LIN {X 0,Y 432.342,Z 838.796,A -85,B 0,C 180,E1 21138.258,E2 21138.258} C_VEL
LIN {X 0,Y 432.858,Z 830.958,A -85,B 0,C 180,E1 21135.431,E2 21135.431} C_VEL
LIN {X 0,Y 433.67,Z 821.606,A -85,B 0,C 180,E1 21132.698,E2 21132.698} C_VEL
LIN {X 0,Y 434.794,Z 810.85,A -85,B 0,C 180,E1 21130.103,E2 21130.103} C_VEL
LIN {X 0,Y 436.206,Z 798.707,A -85,B 0,C 180,E1 21127.636,E2 21127.636} C_VEL
LIN {X 0,Y 437.923,Z 785.326,A -85,B 0,C 180,E1 21125.304,E2 21125.304} C_VEL
LIN {X 0,Y 439.952,Z 770.003,A -85,B 0,C 180,E1 21123.039,E2 21123.039} C_VEL
LIN {X 0,Y 442.141,Z 753.688,A -85,B 0,C 180,E1 21120.984,E2 21120.984} C_VEL
LIN {X 0,Y 444.605,Z 735.27,A -85,B 0,C 180,E1 21119.004,E2 21119.004} C_VEL
LIN {X 0,Y 447.006,Z 716.668,A -85,B 0,C 180,E1 21117.305,E2 21117.305} C_VEL
LIN {X 0,Y 449.34,Z 697.148,A -85,B 0,C 180,E1 21115.817,E2 21115.817} C_VEL
LIN {X 0,Y 451.636,Z 676.412,A -85,B 0,C 180,E1 21114.499,E2 21114.499} C_VEL
LIN {X 0,Y 453.72,Z 655.392,A -85,B 0,C 180,E1 21113.41,E2 21113.41} C_VEL
LIN {X 0,Y 455.533,Z 633.906,A -85,B 0,C 180,E1 21112.542,E2 21112.542} C_VEL
LIN {X 0,Y 456.937,Z 612.319,A -85,B 0,C 180,E1 21111.907,E2 21111.907} C_VEL
LIN {X 0,Y 458.017,Z 582.765,A -85,B 0,C 180,E1 21111.317,E2 21111.317} C_VEL
LIN {X 0,Y 464.099,Z 362.571,A -85,B 0,C 180,E1 21107.412,E2 21107.412} C_VEL
LIN {X 0,Y 464.742,Z 333.232,A -85,B 0,C 180,E1 21106.874,E2 21106.874} C_VEL
LIN {X 0,Y 464.066,Z 331.268,A -85,B 0,C 180,E1 21106.761,E2 21106.761} C_VEL
LIN {X 0,Y 451.341,Z 310.172,A -85,B 0,C 180,E1 21104.898,E2 21104.898} C_VEL
LIN {X 0,Y 448.432,Z 305.591,A -85,B 0,C 180,E1 21104.436,E2 21104.436} C_VEL
LIN {X 0,Y 441.155,Z 290.184,A -85,B 0,C 180,E1 21101.959,E2 21101.959} C_VEL
LIN {X 0,Y 437.067,Z 281.96,A -85,B 0,C 180,E1 21100.518,E2 21100.518} C_VEL
LIN {X 0,Y 434.855,Z 277.707,A -85,B 0,C 180,E1 21099.732,E2 21099.732} C_VEL
LIN {X 0,Y 433.312,Z 274.093,A -85,B 0,C 180,E1 21099.045,E2 21099.045} C_VEL
LIN {X 0,Y 433.24,Z 273.726,A -85,B 0,C 180,E1 21097.204,E2 21097.204} C_VEL
LIN {X 0,Y 433.217,Z 273.762,A -85,B 0,C 180,E1 21093.477,E2 21093.477} C_VEL
LIN {X 0,Y 433.2,Z 273.744,A -85,B 0,C 180,E1 21089.751,E2 21089.751} C_VEL
LIN {X 0,Y 433.199,Z 273.765,A -85,B 0,C 180,E1 21086.01,E2 21086.01} C_VEL
LIN {X 0,Y 433.212,Z 273.763,A -85,B 0,C 180,E1 21082.384,E2 21082.384} C_VEL
LIN {X 0,Y 433.236,Z 273.758,A -85,B 0,C 180,E1 21078.711,E2 21078.711} C_VEL
LIN {X 0,Y 433.233,Z 273.756,A -85,B 0,C 180,E1 21074.843,E2 21074.843} C_VEL
LIN {X 0,Y 433.21,Z 273.757,A -85,B 0,C 180,E1 21071.044,E2 21071.044} C_VEL
LIN {X 0,Y 433.19,Z 273.76,A -85,B 0,C 180,E1 21067.426,E2 21067.426} C_VEL
LIN {X 0,Y 433.193,Z 273.766,A -85,B 0,C 180,E1 21063.705,E2 21063.705} C_VEL
LIN {X 0,Y 433.208,Z 273.769,A -85,B 0,C 180,E1 21060,E2 21060} C_VEL
LIN {X 0,Y 433.236,Z 273.77,A -85,B 0,C 180,E1 21056.295,E2 21056.295} C_VEL
LIN {X 0,Y 433.261,Z 273.765,A -85,B 0,C 180,E1 21052.441,E2 21052.441} C_VEL
LIN {X 0,Y 433.254,Z 273.759,A -85,B 0,C 180,E1 21048.552,E2 21048.552} C_VEL
LIN {X 0,Y 433.255,Z 273.755,A -85,B 0,C 180,E1 21044.715,E2 21044.715} C_VEL
LIN {X 0,Y 433.234,Z 273.756,A -85,B 0,C 180,E1 21041.009,E2 21041.009} C_VEL
LIN {X 0,Y 433.226,Z 273.756,A -85,B 0,C 180,E1 21037.33,E2 21037.33} C_VEL
LIN {X 0,Y 433.232,Z 273.757,A -85,B 0,C 180,E1 21033.549,E2 21033.549} C_VEL
LIN {X 0,Y 433.252,Z 273.729,A -85,B 0,C 180,E1 21029.928,E2 21029.928} C_VEL
LIN {X 0,Y 433.259,Z 273.766,A -85,B 0,C 180,E1 21026.049,E2 21026.049} C_VEL
LIN {X 0,Y 433.251,Z 273.723,A -85,B 0,C 180,E1 21022.297,E2 21022.297} C_VEL
LIN {X 0,Y 433.255,Z 273.731,A -85,B 0,C 180,E1 21018.522,E2 21018.522} C_VEL
LIN {X 0,Y 433.329,Z 274.222,A -85,B 0,C 180,E1 21017.773,E2 21017.773} C_VEL
LIN {X 0,Y 434.815,Z 277.61,A -85,B 0,C 180,E1 21017.105,E2 21017.105} C_VEL
LIN {X 0,Y 441.185,Z 290.862,A -85,B 0,C 180,E1 21014.631,E2 21014.631} C_VEL
LIN {X 0,Y 448.978,Z 308.721,A -85,B 0,C 180,E1 21011.656,E2 21011.656} C_VEL
LIN {X 0,Y 455.647,Z 325.683,A -85,B 0,C 180,E1 21009.149,E2 21009.149} C_VEL
LIN {X 0,Y 461.307,Z 360.167,A -85,B 0,C 180,E1 21007.848,E2 21007.848} C_VEL
LIN {X 0,Y 457.058,Z 564.663,A -85,B 0,C 180,E1 21004.513,E2 21004.513} C_VEL
LIN {X 0,Y 456.111,Z 572.366,A -85,B 0,C 180,E1 21004.467,E2 21004.467} C_VEL
LIN {X 0,Y 450.547,Z 592.852,A -85,B 0,C 180,E1 21004.59,E2 21004.59} C_VEL
LIN {X 0,Y 449.686,Z 599.4,A -85,B 0,C 180,E1 21004.491,E2 21004.491} C_VEL
LIN {X 0,Y 448.443,Z 619.453,A -85,B 0,C 180,E1 21003.895,E2 21003.895} C_VEL
LIN {X 0,Y 446.74,Z 639.526,A -85,B 0,C 180,E1 21003.061,E2 21003.061} C_VEL
LIN {X 0,Y 444.586,Z 659.236,A -85,B 0,C 180,E1 21001.98,E2 21001.98} C_VEL
LIN {X 0,Y 442.233,Z 677.397,A -85,B 0,C 180,E1 21000.728,E2 21000.728} C_VEL
LIN {X 0,Y 439.717,Z 694.787,A -85,B 0,C 180,E1 20999.266,E2 20999.266} C_VEL
LIN {X 0,Y 437.101,Z 711.358,A -85,B 0,C 180,E1 20997.594,E2 20997.594} C_VEL
LIN {X 0,Y 434.515,Z 726.984,A -85,B 0,C 180,E1 20995.709,E2 20995.709} C_VEL
LIN {X 0,Y 431.994,Z 741.73,A -85,B 0,C 180,E1 20993.573,E2 20993.573} C_VEL
LIN {X 0,Y 429.869,Z 754.225,A -85,B 0,C 180,E1 20991.418,E2 20991.418} C_VEL
LIN {X 0,Y 427.951,Z 766.244,A -85,B 0,C 180,E1 20988.95,E2 20988.95} C_VEL
LIN {X 0,Y 426.43,Z 776.74,A -85,B 0,C 180,E1 20986.341,E2 20986.341} C_VEL
LIN {X 0,Y 425.369,Z 785.323,A -85,B 0,C 180,E1 20983.733,E2 20983.733} C_VEL
LIN {X 0,Y 424.64,Z 792.647,A -85,B 0,C 180,E1 20980.926,E2 20980.926} C_VEL
LIN {X 0,Y 424.24,Z 798.109,A -85,B 0,C 180,E1 20978.129,E2 20978.129} C_VEL
LIN {X 0,Y 424.047,Z 801.843,A -85,B 0,C 180,E1 20975.412,E2 20975.412} C_VEL
LIN {X 0,Y 423.984,Z 804.16,A -85,B 0,C 180,E1 20972.568,E2 20972.568} C_VEL
LIN {X 0,Y 423.977,Z 804.889,A -85,B 0,C 180,E1 20969.865,E2 20969.865} C_VEL
LIN {X 0,Y 423.986,Z 804.012,A -85,B 0,C 180,E1 20967.026,E2 20967.026} C_VEL
LIN {X 0,Y 424.055,Z 801.599,A -85,B 0,C 180,E1 20964.278,E2 20964.278} C_VEL
LIN {X 0,Y 424.272,Z 797.547,A -85,B 0,C 180,E1 20961.462,E2 20961.462} C_VEL
LIN {X 0,Y 424.687,Z 792.034,A -85,B 0,C 180,E1 20958.732,E2 20958.732} C_VEL
LIN {X 0,Y 425.429,Z 784.801,A -85,B 0,C 180,E1 20955.991,E2 20955.991} C_VEL
LIN {X 0,Y 426.596,Z 775.591,A -85,B 0,C 180,E1 20953.245,E2 20953.245} C_VEL
LIN {X 0,Y 428.083,Z 765.421,A -85,B 0,C 180,E1 20950.773,E2 20950.773} C_VEL
LIN {X 0,Y 429.914,Z 753.959,A -85,B 0,C 180,E1 20948.441,E2 20948.441} C_VEL
LIN {X 0,Y 432.079,Z 741.214,A -85,B 0,C 180,E1 20946.257,E2 20946.257} C_VEL
LIN {X 0,Y 434.58,Z 726.625,A -85,B 0,C 180,E1 20944.152,E2 20944.152} C_VEL
LIN {X 0,Y 437.285,Z 710.326,A -85,B 0,C 180,E1 20942.197,E2 20942.197} C_VEL
LIN {X 0,Y 439.941,Z 693.383,A -85,B 0,C 180,E1 20940.511,E2 20940.511} C_VEL
LIN {X 0,Y 442.454,Z 675.834,A -85,B 0,C 180,E1 20939.063,E2 20939.063} C_VEL
LIN {X 0,Y 444.822,Z 657.259,A -85,B 0,C 180,E1 20937.811,E2 20937.811} C_VEL
LIN {X 0,Y 446.807,Z 638.92,A -85,B 0,C 180,E1 20936.818,E2 20936.818} C_VEL
LIN {X 0,Y 448.538,Z 618.51,A -85,B 0,C 180,E1 20935.979,E2 20935.979} C_VEL
LIN {X 0,Y 449.739,Z 598.65,A -85,B 0,C 180,E1 20935.398,E2 20935.398} C_VEL
LIN {X 0,Y 450.572,Z 571.156,A -85,B 0,C 180,E1 20934.885,E2 20934.885} C_VEL
LIN {X 0,Y 455.175,Z 360.498,A -85,B 0,C 180,E1 20931.4,E2 20931.4} C_VEL
LIN {X 0,Y 449.82,Z 329.343,A -85,B 0,C 180,E1 20930.173,E2 20930.173} C_VEL
LIN {X 0,Y 447.126,Z 324.378,A -85,B 0,C 180,E1 20929.689,E2 20929.689} C_VEL
LIN {X 0,Y 440.044,Z 306.845,A -85,B 0,C 180,E1 20926.929,E2 20926.929} C_VEL
LIN {X 0,Y 433.12,Z 291.369,A -85,B 0,C 180,E1 20924.201,E2 20924.201} C_VEL
LIN {X 0,Y 428.555,Z 282.138,A -85,B 0,C 180,E1 20922.397,E2 20922.397} C_VEL
LIN {X 0,Y 426.709,Z 278.339,A -85,B 0,C 180,E1 20921.63,E2 20921.63} C_VEL
LIN {X 0,Y 425.329,Z 274.888,A -85,B 0,C 180,E1 20920.864,E2 20920.864} C_VEL
LIN {X 0,Y 425.309,Z 274.709,A -85,B 0,C 180,E1 20917.162,E2 20917.162} C_VEL
LIN {X 0,Y 425.316,Z 274.741,A -85,B 0,C 180,E1 20913.374,E2 20913.374} C_VEL
LIN {X 0,Y 425.317,Z 274.725,A -85,B 0,C 180,E1 20909.566,E2 20909.566} C_VEL
LIN {X 0,Y 425.318,Z 274.743,A -85,B 0,C 180,E1 20905.78,E2 20905.78} C_VEL
LIN {X 0,Y 425.314,Z 274.743,A -85,B 0,C 180,E1 20901.95,E2 20901.95} C_VEL
LIN {X 0,Y 425.292,Z 274.744,A -85,B 0,C 180,E1 20898.221,E2 20898.221} C_VEL
LIN {X 0,Y 425.282,Z 274.743,A -85,B 0,C 180,E1 20894.395,E2 20894.395} C_VEL
LIN {X 0,Y 425.278,Z 274.742,A -85,B 0,C 180,E1 20890.567,E2 20890.567} C_VEL
LIN {X 0,Y 425.28,Z 274.748,A -85,B 0,C 180,E1 20886.751,E2 20886.751} C_VEL
LIN {X 0,Y 425.289,Z 274.754,A -85,B 0,C 180,E1 20882.965,E2 20882.965} C_VEL
LIN {X 0,Y 425.307,Z 274.759,A -85,B 0,C 180,E1 20879.192,E2 20879.192} C_VEL
LIN {X 0,Y 425.304,Z 274.757,A -85,B 0,C 180,E1 20875.28,E2 20875.28} C_VEL
LIN {X 0,Y 425.293,Z 274.751,A -85,B 0,C 180,E1 20871.483,E2 20871.483} C_VEL
LIN {X 0,Y 425.27,Z 274.749,A -85,B 0,C 180,E1 20867.646,E2 20867.646} C_VEL
LIN {X 0,Y 425.241,Z 274.748,A -85,B 0,C 180,E1 20864.032,E2 20864.032} C_VEL
LIN {X 0,Y 425.247,Z 274.75,A -85,B 0,C 180,E1 20860.21,E2 20860.21} C_VEL
LIN {X 0,Y 425.256,Z 274.752,A -85,B 0,C 180,E1 20856.441,E2 20856.441} C_VEL
LIN {X 0,Y 425.28,Z 274.753,A -85,B 0,C 180,E1 20852.707,E2 20852.707} C_VEL
LIN {X 0,Y 425.309,Z 274.707,A -85,B 0,C 180,E1 20849.013,E2 20849.013} C_VEL
LIN {X 0,Y 425.312,Z 274.742,A -85,B 0,C 180,E1 20845.128,E2 20845.128} C_VEL
LIN {X 0,Y 425.305,Z 274.978,A -85,B 0,C 180,E1 20842.151,E2 20842.151} C_VEL
LIN {X 0,Y 426.746,Z 278.433,A -85,B 0,C 180,E1 20841.448,E2 20841.448} C_VEL
LIN {X 0,Y 427.86,Z 280.355,A -85,B 0,C 180,E1 20841.052,E2 20841.052} C_VEL
LIN {X 0,Y 434.06,Z 292.497,A -85,B 0,C 180,E1 20838.792,E2 20838.792} C_VEL
LIN {X 0,Y 440.782,Z 306.575,A -85,B 0,C 180,E1 20836.47,E2 20836.47} C_VEL
LIN {X 0,Y 453.474,Z 326.821,A -85,B 0,C 180,E1 20834.498,E2 20834.498} C_VEL
LIN {X 0,Y 458.777,Z 336.288,A -85,B 0,C 180,E1 20833.704,E2 20833.704} C_VEL
LIN {X 0,Y 452.487,Z 549.122,A -85,B 0,C 180,E1 20829.882,E2 20829.882} C_VEL
LIN {X 0,Y 450.683,Z 607.462,A -85,B 0,C 180,E1 20828.803,E2 20828.803} C_VEL
LIN {X 0,Y 449.222,Z 629.594,A -85,B 0,C 180,E1 20828.179,E2 20828.179} C_VEL
LIN {X 0,Y 447.415,Z 650.894,A -85,B 0,C 180,E1 20827.351,E2 20827.351} C_VEL
LIN {X 0,Y 445.277,Z 671.891,A -85,B 0,C 180,E1 20826.307,E2 20826.307} C_VEL
LIN {X 0,Y 442.975,Z 691.862,A -85,B 0,C 180,E1 20825.067,E2 20825.067} C_VEL
LIN {X 0,Y 440.506,Z 711.034,A -85,B 0,C 180,E1 20823.629,E2 20823.629} C_VEL
LIN {X 0,Y 437.891,Z 730.422,A -85,B 0,C 180,E1 20821.91,E2 20821.91} C_VEL
LIN {X 0,Y 435.415,Z 748.423,A -85,B 0,C 180,E1 20820.036,E2 20820.036} C_VEL
LIN {X 0,Y 432.988,Z 765.307,A -85,B 0,C 180,E1 20817.954,E2 20817.954} C_VEL
LIN {X 0,Y 430.798,Z 780.808,A -85,B 0,C 180,E1 20815.722,E2 20815.722} C_VEL
LIN {X 0,Y 429.003,Z 794.229,A -85,B 0,C 180,E1 20813.486,E2 20813.486} C_VEL
LIN {X 0,Y 427.37,Z 806.957,A -85,B 0,C 180,E1 20810.974,E2 20810.974} C_VEL
LIN {X 0,Y 426.071,Z 818.284,A -85,B 0,C 180,E1 20808.328,E2 20808.328} C_VEL
LIN {X 0,Y 425.154,Z 827.798,A -85,B 0,C 180,E1 20805.691,E2 20805.691} C_VEL
LIN {X 0,Y 424.519,Z 835.821,A -85,B 0,C 180,E1 20802.929,E2 20802.929} C_VEL
LIN {X 0,Y 424.146,Z 842.478,A -85,B 0,C 180,E1 20800.046,E2 20800.046} C_VEL
LIN {X 0,Y 423.986,Z 847.207,A -85,B 0,C 180,E1 20797.316,E2 20797.316} C_VEL
LIN {X 0,Y 423.922,Z 850.344,A -85,B 0,C 180,E1 20794.599,E2 20794.599} C_VEL
LIN {X 0,Y 423.903,Z 852.117,A -85,B 0,C 180,E1 20791.892,E2 20791.892} C_VEL
LIN {X 0,Y 423.905,Z 852.344,A -85,B 0,C 180,E1 20789.189,E2 20789.189} C_VEL
LIN {X 0,Y 423.911,Z 851.265,A -85,B 0,C 180,E1 20786.484,E2 20786.484} C_VEL
LIN {X 0,Y 423.945,Z 848.609,A -85,B 0,C 180,E1 20783.772,E2 20783.772} C_VEL
LIN {X 0,Y 424.056,Z 844.592,A -85,B 0,C 180,E1 20781.048,E2 20781.048} C_VEL
LIN {X 0,Y 424.332,Z 838.905,A -85,B 0,C 180,E1 20778.309,E2 20778.309} C_VEL
LIN {X 0,Y 424.859,Z 831.189,A -85,B 0,C 180,E1 20775.416,E2 20775.416} C_VEL
LIN {X 0,Y 425.69,Z 822.043,A -85,B 0,C 180,E1 20772.645,E2 20772.645} C_VEL
LIN {X 0,Y 426.888,Z 811.022,A -85,B 0,C 180,E1 20769.921,E2 20769.921} C_VEL
LIN {X 0,Y 428.404,Z 798.659,A -85,B 0,C 180,E1 20767.351,E2 20767.351} C_VEL
LIN {X 0,Y 430.206,Z 785.265,A -85,B 0,C 180,E1 20764.977,E2 20764.977} C_VEL
LIN {X 0,Y 432.265,Z 770.439,A -85,B 0,C 180,E1 20762.744,E2 20762.744} C_VEL
LIN {X 0,Y 434.634,Z 753.687,A -85,B 0,C 180,E1 20760.585,E2 20760.585} C_VEL
LIN {X 0,Y 437.135,Z 736.043,A -85,B 0,C 180,E1 20758.645,E2 20758.645} C_VEL
LIN {X 0,Y 439.757,Z 716.905,A -85,B 0,C 180,E1 20756.852,E2 20756.852} C_VEL
LIN {X 0,Y 442.22,Z 697.805,A -85,B 0,C 180,E1 20755.353,E2 20755.353} C_VEL
LIN {X 0,Y 444.704,Z 676.971,A -85,B 0,C 180,E1 20753.99,E2 20753.99} C_VEL
LIN {X 0,Y 446.923,Z 656.118,A -85,B 0,C 180,E1 20752.881,E2 20752.881} C_VEL
LIN {X 0,Y 448.807,Z 634.988,A -85,B 0,C 180,E1 20752.008,E2 20752.008} C_VEL
LIN {X 0,Y 450.335,Z 613.288,A -85,B 0,C 180,E1 20751.347,E2 20751.347} C_VEL
LIN {X 0,Y 451.401,Z 587.981,A -85,B 0,C 180,E1 20750.816,E2 20750.816} C_VEL
LIN {X 0,Y 457.893,Z 365.769,A -85,B 0,C 180,E1 20746.824,E2 20746.824} C_VEL
LIN {X 0,Y 458.663,Z 335.761,A -85,B 0,C 180,E1 20746.273,E2 20746.273} C_VEL
LIN {X 0,Y 446.377,Z 315.309,A -85,B 0,C 180,E1 20744.425,E2 20744.425} C_VEL
LIN {X 0,Y 440.405,Z 305.946,A -85,B 0,C 180,E1 20743.464,E2 20743.464} C_VEL
LIN {X 0,Y 433.548,Z 291.624,A -85,B 0,C 180,E1 20741.052,E2 20741.052} C_VEL
LIN {X 0,Y 428.845,Z 282.534,A -85,B 0,C 180,E1 20739.358,E2 20739.358} C_VEL
LIN {X 0,Y 427.13,Z 278.929,A -85,B 0,C 180,E1 20738.683,E2 20738.683} C_VEL
LIN {X 0,Y 425.432,Z 275.615,A -85,B 0,C 180,E1 20738.007,E2 20738.007} C_VEL
LIN {X 0,Y 425.301,Z 274.942,A -85,B 0,C 180,E1 20737.824,E2 20737.824} C_VEL
LIN {X 0,Y 425.283,Z 274.761,A -85,B 0,C 180,E1 20734.35,E2 20734.35} C_VEL
LIN {X 0,Y 425.296,Z 274.711,A -85,B 0,C 180,E1 20730.635,E2 20730.635} C_VEL
LIN {X 0,Y 425.308,Z 274.746,A -85,B 0,C 180,E1 20726.832,E2 20726.832} C_VEL
LIN {X 0,Y 425.299,Z 274.745,A -85,B 0,C 180,E1 20722.97,E2 20722.97} C_VEL
LIN {X 0,Y 425.268,Z 274.746,A -85,B 0,C 180,E1 20719.217,E2 20719.217} C_VEL
LIN {X 0,Y 425.244,Z 274.747,A -85,B 0,C 180,E1 20715.548,E2 20715.548} C_VEL
LIN {X 0,Y 425.241,Z 274.748,A -85,B 0,C 180,E1 20711.804,E2 20711.804} C_VEL
LIN {X 0,Y 425.26,Z 274.752,A -85,B 0,C 180,E1 20708.11,E2 20708.11} C_VEL
LIN {X 0,Y 425.294,Z 274.755,A -85,B 0,C 180,E1 20704.449,E2 20704.449} C_VEL
LIN {X 0,Y 425.313,Z 274.757,A -85,B 0,C 180,E1 20700.539,E2 20700.539} C_VEL
LIN {X 0,Y 425.308,Z 274.757,A -85,B 0,C 180,E1 20696.63,E2 20696.63} C_VEL
LIN {X 0,Y 425.314,Z 274.75,A -85,B 0,C 180,E1 20692.707,E2 20692.707} C_VEL
LIN {X 0,Y 425.296,Z 274.745,A -85,B 0,C 180,E1 20688.885,E2 20688.885} C_VEL
LIN {X 0,Y 425.282,Z 274.744,A -85,B 0,C 180,E1 20685.151,E2 20685.151} C_VEL
LIN {X 0,Y 425.284,Z 274.744,A -85,B 0,C 180,E1 20681.341,E2 20681.341} C_VEL
LIN {X 0,Y 425.287,Z 274.744,A -85,B 0,C 180,E1 20677.467,E2 20677.467} C_VEL
LIN {X 0,Y 425.296,Z 274.744,A -85,B 0,C 180,E1 20673.619,E2 20673.619} C_VEL
LIN {X 0,Y 425.311,Z 274.714,A -85,B 0,C 180,E1 20669.894,E2 20669.894} C_VEL
LIN {X 0,Y 425.317,Z 274.756,A -85,B 0,C 180,E1 20665.978,E2 20665.978} C_VEL
LIN {X 0,Y 425.313,Z 274.711,A -85,B 0,C 180,E1 20662.151,E2 20662.151} C_VEL
LIN {X 0,Y 425.338,Z 274.956,A -85,B 0,C 180,E1 20658.987,E2 20658.987} C_VEL
LIN {X 0,Y 426.671,Z 278.285,A -85,B 0,C 180,E1 20658.277,E2 20658.277} C_VEL
LIN {X 0,Y 431.664,Z 288.3,A -85,B 0,C 180,E1 20656.275,E2 20656.275} C_VEL
LIN {X 0,Y 438.677,Z 303.743,A -85,B 0,C 180,E1 20653.497,E2 20653.497} C_VEL
LIN {X 0,Y 445.468,Z 320.179,A -85,B 0,C 180,E1 20650.852,E2 20650.852} C_VEL
LIN {X 0,Y 447.868,Z 326.008,A -85,B 0,C 180,E1 20650.027,E2 20650.027} C_VEL
LIN {X 0,Y 450.129,Z 330.276,A -85,B 0,C 180,E1 20649.675,E2 20649.675} C_VEL
LIN {X 0,Y 455.193,Z 361.696,A -85,B 0,C 180,E1 20648.477,E2 20648.477} C_VEL
LIN {X 0,Y 449.956,Z 594.214,A -85,B 0,C 180,E1 20644.617,E2 20644.617} C_VEL
LIN {X 0,Y 449.686,Z 599.4,A -85,B 0,C 180,E1 20644.491,E2 20644.491} C_VEL
LIN {X 0,Y 448.171,Z 608.086,A -85,B 0,C 180,E1 20644.363,E2 20644.363} C_VEL
LIN {X 0,Y 442.571,Z 625.029,A -85,B 0,C 180,E1 20644.211,E2 20644.211} C_VEL
LIN {X 0,Y 440.918,Z 632.44,A -85,B 0,C 180,E1 20643.996,E2 20643.996} C_VEL
LIN {X 0,Y 440.796,Z 633.461,A -85,B 0,C 180,E1 20643.953,E2 20643.953} C_VEL
LIN {X 0,Y 438.804,Z 652.395,A -85,B 0,C 180,E1 20642.995,E2 20642.995} C_VEL
LIN {X 0,Y 436.421,Z 671.242,A -85,B 0,C 180,E1 20641.79,E2 20641.79} C_VEL
LIN {X 0,Y 433.688,Z 689.657,A -85,B 0,C 180,E1 20640.324,E2 20640.324} C_VEL
LIN {X 0,Y 430.962,Z 706.412,A -85,B 0,C 180,E1 20638.701,E2 20638.701} C_VEL
LIN {X 0,Y 428.095,Z 722.858,A -85,B 0,C 180,E1 20636.792,E2 20636.792} C_VEL
LIN {X 0,Y 425.43,Z 737.71,A -85,B 0,C 180,E1 20634.729,E2 20634.729} C_VEL
LIN {X 0,Y 423.03,Z 751.127,A -85,B 0,C 180,E1 20632.513,E2 20632.513} C_VEL
LIN {X 0,Y 420.834,Z 763.774,A -85,B 0,C 180,E1 20630.006,E2 20630.006} C_VEL
LIN {X 0,Y 419.054,Z 774.772,A -85,B 0,C 180,E1 20627.352,E2 20627.352} C_VEL
LIN {X 0,Y 417.782,Z 783.758,A -85,B 0,C 180,E1 20624.695,E2 20624.695} C_VEL
LIN {X 0,Y 416.886,Z 791.376,A -85,B 0,C 180,E1 20621.888,E2 20621.888} C_VEL
LIN {X 0,Y 416.366,Z 797.415,A -85,B 0,C 180,E1 20618.98,E2 20618.98} C_VEL
LIN {X 0,Y 416.119,Z 801.567,A -85,B 0,C 180,E1 20616.207,E2 20616.207} C_VEL
LIN {X 0,Y 416.009,Z 804.256,A -85,B 0,C 180,E1 20613.307,E2 20613.307} C_VEL
LIN {X 0,Y 415.982,Z 805.258,A -85,B 0,C 180,E1 20610.551,E2 20610.551} C_VEL
LIN {X 0,Y 415.992,Z 804.785,A -85,B 0,C 180,E1 20607.658,E2 20607.658} C_VEL
LIN {X 0,Y 416.059,Z 802.871,A -85,B 0,C 180,E1 20604.899,E2 20604.899} C_VEL
LIN {X 0,Y 416.248,Z 799.229,A -85,B 0,C 180,E1 20601.992,E2 20601.992} C_VEL
LIN {X 0,Y 416.638,Z 794.079,A -85,B 0,C 180,E1 20599.212,E2 20599.212} C_VEL
LIN {X 0,Y 417.349,Z 787.26,A -85,B 0,C 180,E1 20596.422,E2 20596.422} C_VEL
LIN {X 0,Y 418.488,Z 778.588,A -85,B 0,C 180,E1 20593.625,E2 20593.625} C_VEL
LIN {X 0,Y 420.053,Z 768.416,A -85,B 0,C 180,E1 20590.968,E2 20590.968} C_VEL
LIN {X 0,Y 422.031,Z 756.769,A -85,B 0,C 180,E1 20588.456,E2 20588.456} C_VEL
LIN {X 0,Y 424.425,Z 743.434,A -85,B 0,C 180,E1 20586.072,E2 20586.072} C_VEL
LIN {X 0,Y 427.061,Z 728.752,A -85,B 0,C 180,E1 20583.887,E2 20583.887} C_VEL
LIN {X 0,Y 429.773,Z 713.364,A -85,B 0,C 180,E1 20581.97,E2 20581.97} C_VEL
LIN {X 0,Y 432.621,Z 696.412,A -85,B 0,C 180,E1 20580.206,E2 20580.206} C_VEL
LIN {X 0,Y 435.317,Z 678.927,A -85,B 0,C 180,E1 20578.697,E2 20578.697} C_VEL
LIN {X 0,Y 437.856,Z 660.443,A -85,B 0,C 180,E1 20577.391,E2 20577.391} C_VEL
LIN {X 0,Y 440.031,Z 641.486,A -85,B 0,C 180,E1 20576.33,E2 20576.33} C_VEL
LIN {X 0,Y 441.83,Z 621.78,A -85,B 0,C 180,E1 20575.477,E2 20575.477} C_VEL
LIN {X 0,Y 443.254,Z 600.889,A -85,B 0,C 180,E1 20574.828,E2 20574.828} C_VEL
LIN {X 0,Y 444.096,Z 578.129,A -85,B 0,C 180,E1 20574.37,E2 20574.37} C_VEL
LIN {X 0,Y 449.135,Z 362.019,A -85,B 0,C 180,E1 20570.754,E2 20570.754} C_VEL
LIN {X 0,Y 444.346,Z 333.544,A -85,B 0,C 180,E1 20569.613,E2 20569.613} C_VEL
LIN {X 0,Y 439.058,Z 324.277,A -85,B 0,C 180,E1 20568.721,E2 20568.721} C_VEL
LIN {X 0,Y 432.276,Z 307.715,A -85,B 0,C 180,E1 20566.001,E2 20566.001} C_VEL
LIN {X 0,Y 425.286,Z 292.398,A -85,B 0,C 180,E1 20563.169,E2 20563.169} C_VEL
LIN {X 0,Y 420.839,Z 283.447,A -85,B 0,C 180,E1 20561.338,E2 20561.338} C_VEL
LIN {X 0,Y 418.859,Z 279.471,A -85,B 0,C 180,E1 20560.489,E2 20560.489} C_VEL
LIN {X 0,Y 417.4,Z 275.929,A -85,B 0,C 180,E1 20559.677,E2 20559.677} C_VEL
LIN {X 0,Y 417.375,Z 275.708,A -85,B 0,C 180,E1 20555.935,E2 20555.935} C_VEL
LIN {X 0,Y 417.371,Z 275.697,A -85,B 0,C 180,E1 20552.129,E2 20552.129} C_VEL
LIN {X 0,Y 417.367,Z 275.747,A -85,B 0,C 180,E1 20548.316,E2 20548.316} C_VEL
LIN {X 0,Y 417.357,Z 275.748,A -85,B 0,C 180,E1 20544.448,E2 20544.448} C_VEL
LIN {X 0,Y 417.354,Z 275.749,A -85,B 0,C 180,E1 20540.62,E2 20540.62} C_VEL
LIN {X 0,Y 417.349,Z 275.75,A -85,B 0,C 180,E1 20536.708,E2 20536.708} C_VEL
LIN {X 0,Y 417.353,Z 275.747,A -85,B 0,C 180,E1 20532.874,E2 20532.874} C_VEL
LIN {X 0,Y 417.363,Z 275.736,A -85,B 0,C 180,E1 20529.098,E2 20529.098} C_VEL
LIN {X 0,Y 417.374,Z 275.729,A -85,B 0,C 180,E1 20525.361,E2 20525.361} C_VEL
LIN {X 0,Y 417.369,Z 275.729,A -85,B 0,C 180,E1 20521.51,E2 20521.51} C_VEL
LIN {X 0,Y 417.34,Z 275.737,A -85,B 0,C 180,E1 20517.803,E2 20517.803} C_VEL
LIN {X 0,Y 417.321,Z 275.749,A -85,B 0,C 180,E1 20514.087,E2 20514.087} C_VEL
LIN {X 0,Y 417.311,Z 275.752,A -85,B 0,C 180,E1 20510.345,E2 20510.345} C_VEL
LIN {X 0,Y 417.311,Z 275.752,A -85,B 0,C 180,E1 20506.561,E2 20506.561} C_VEL
LIN {X 0,Y 417.329,Z 275.749,A -85,B 0,C 180,E1 20502.861,E2 20502.861} C_VEL
LIN {X 0,Y 417.359,Z 275.745,A -85,B 0,C 180,E1 20499.087,E2 20499.087} C_VEL
LIN {X 0,Y 417.363,Z 275.749,A -85,B 0,C 180,E1 20495.214,E2 20495.214} C_VEL
LIN {X 0,Y 417.371,Z 275.741,A -85,B 0,C 180,E1 20491.255,E2 20491.255} C_VEL
LIN {X 0,Y 417.346,Z 275.708,A -85,B 0,C 180,E1 20487.488,E2 20487.488} C_VEL
LIN {X 0,Y 417.338,Z 275.74,A -85,B 0,C 180,E1 20483.718,E2 20483.718} C_VEL
LIN {X 0,Y 417.47,Z 276.341,A -85,B 0,C 180,E1 20483.266,E2 20483.266} C_VEL
LIN {X 0,Y 419.119,Z 279.84,A -85,B 0,C 180,E1 20482.531,E2 20482.531} C_VEL
LIN {X 0,Y 422.59,Z 286.572,A -85,B 0,C 180,E1 20481.171,E2 20481.171} C_VEL
LIN {X 0,Y 428.388,Z 297.927,A -85,B 0,C 180,E1 20479.016,E2 20479.016} C_VEL
LIN {X 0,Y 432.651,Z 306.855,A -85,B 0,C 180,E1 20477.511,E2 20477.511} C_VEL
LIN {X 0,Y 445.037,Z 326.238,A -85,B 0,C 180,E1 20475.496,E2 20475.496} C_VEL
LIN {X 0,Y 452.67,Z 339.479,A -85,B 0,C 180,E1 20474.315,E2 20474.315} C_VEL
LIN {X 0,Y 446.088,Z 550.51,A -85,B 0,C 180,E1 20470.48,E2 20470.48} C_VEL
LIN {X 0,Y 444.229,Z 607.33,A -85,B 0,C 180,E1 20469.413,E2 20469.413} C_VEL
LIN {X 0,Y 442.691,Z 629.472,A -85,B 0,C 180,E1 20468.782,E2 20468.782} C_VEL
LIN {X 0,Y 440.763,Z 651.005,A -85,B 0,C 180,E1 20467.933,E2 20467.933} C_VEL
LIN {X 0,Y 438.557,Z 671.563,A -85,B 0,C 180,E1 20466.896,E2 20466.896} C_VEL
LIN {X 0,Y 436.072,Z 691.87,A -85,B 0,C 180,E1 20465.618,E2 20465.618} C_VEL
LIN {X 0,Y 433.479,Z 710.831,A -85,B 0,C 180,E1 20464.169,E2 20464.169} C_VEL
LIN {X 0,Y 430.704,Z 730.058,A -85,B 0,C 180,E1 20462.428,E2 20462.428} C_VEL
LIN {X 0,Y 427.965,Z 748.573,A -85,B 0,C 180,E1 20460.447,E2 20460.447} C_VEL
LIN {X 0,Y 425.274,Z 766.36,A -85,B 0,C 180,E1 20458.2,E2 20458.2} C_VEL
LIN {X 0,Y 422.994,Z 781.631,A -85,B 0,C 180,E1 20455.931,E2 20455.931} C_VEL
LIN {X 0,Y 421.016,Z 795.593,A -85,B 0,C 180,E1 20453.514,E2 20453.514} C_VEL
LIN {X 0,Y 419.36,Z 808.181,A -85,B 0,C 180,E1 20450.955,E2 20450.955} C_VEL
LIN {X 0,Y 418.042,Z 819.255,A -85,B 0,C 180,E1 20448.259,E2 20448.259} C_VEL
LIN {X 0,Y 417.081,Z 828.917,A -85,B 0,C 180,E1 20445.432,E2 20445.432} C_VEL
LIN {X 0,Y 416.464,Z 836.753,A -85,B 0,C 180,E1 20442.619,E2 20442.619} C_VEL
LIN {X 0,Y 416.13,Z 842.766,A -85,B 0,C 180,E1 20439.822,E2 20439.822} C_VEL
LIN {X 0,Y 415.977,Z 847.473,A -85,B 0,C 180,E1 20436.902,E2 20436.902} C_VEL
LIN {X 0,Y 415.926,Z 850.236,A -85,B 0,C 180,E1 20434.274,E2 20434.274} C_VEL
LIN {X 0,Y 415.916,Z 851.802,A -85,B 0,C 180,E1 20431.377,E2 20431.377} C_VEL
LIN {X 0,Y 415.919,Z 851.826,A -85,B 0,C 180,E1 20428.76,E2 20428.76} C_VEL
LIN {X 0,Y 415.923,Z 850.354,A -85,B 0,C 180,E1 20425.864,E2 20425.864} C_VEL
LIN {X 0,Y 415.968,Z 847.638,A -85,B 0,C 180,E1 20423.236,E2 20423.236} C_VEL
LIN {X 0,Y 416.121,Z 843.039,A -85,B 0,C 180,E1 20420.317,E2 20420.317} C_VEL
LIN {X 0,Y 416.443,Z 837.104,A -85,B 0,C 180,E1 20417.521,E2 20417.521} C_VEL
LIN {X 0,Y 417.042,Z 829.343,A -85,B 0,C 180,E1 20414.709,E2 20414.709} C_VEL
LIN {X 0,Y 417.986,Z 819.796,A -85,B 0,C 180,E1 20411.883,E2 20411.883} C_VEL
LIN {X 0,Y 419.28,Z 808.837,A -85,B 0,C 180,E1 20409.187,E2 20409.187} C_VEL
LIN {X 0,Y 420.911,Z 796.348,A -85,B 0,C 180,E1 20406.629,E2 20406.629} C_VEL
LIN {X 0,Y 422.995,Z 781.648,A -85,B 0,C 180,E1 20404.069,E2 20404.069} C_VEL
LIN {X 0,Y 425.276,Z 766.368,A -85,B 0,C 180,E1 20401.8,E2 20401.8} C_VEL
LIN {X 0,Y 427.966,Z 748.572,A -85,B 0,C 180,E1 20399.552,E2 20399.552} C_VEL
LIN {X 0,Y 430.705,Z 730.059,A -85,B 0,C 180,E1 20397.572,E2 20397.572} C_VEL
LIN {X 0,Y 433.479,Z 710.833,A -85,B 0,C 180,E1 20395.831,E2 20395.831} C_VEL
LIN {X 0,Y 436.191,Z 690.835,A -85,B 0,C 180,E1 20394.313,E2 20394.313} C_VEL
LIN {X 0,Y 438.756,Z 670.028,A -85,B 0,C 180,E1 20393.015,E2 20393.015} C_VEL
LIN {X 0,Y 440.986,Z 648.747,A -85,B 0,C 180,E1 20391.966,E2 20391.966} C_VEL
LIN {X 0,Y 442.902,Z 626.421,A -85,B 0,C 180,E1 20391.12,E2 20391.12} C_VEL
LIN {X 0,Y 444.377,Z 604.158,A -85,B 0,C 180,E1 20390.521,E2 20390.521} C_VEL
LIN {X 0,Y 450.904,Z 395.819,A -85,B 0,C 180,E1 20386.708,E2 20386.708} C_VEL
LIN {X 0,Y 452.564,Z 339.015,A -85,B 0,C 180,E1 20385.665,E2 20385.665} C_VEL
LIN {X 0,Y 440.669,Z 319.242,A -85,B 0,C 180,E1 20383.819,E2 20383.819} C_VEL
LIN {X 0,Y 432.233,Z 306.09,A -85,B 0,C 180,E1 20382.4,E2 20382.4} C_VEL
LIN {X 0,Y 425.42,Z 292.132,A -85,B 0,C 180,E1 20379.913,E2 20379.913} C_VEL
LIN {X 0,Y 421.536,Z 284.405,A -85,B 0,C 180,E1 20378.422,E2 20378.422} C_VEL
LIN {X 0,Y 418.695,Z 279.242,A -85,B 0,C 180,E1 20377.341,E2 20377.341} C_VEL
LIN {X 0,Y 417.39,Z 275.942,A -85,B 0,C 180,E1 20376.618,E2 20376.618} C_VEL
LIN {X 0,Y 417.371,Z 275.714,A -85,B 0,C 180,E1 20372.943,E2 20372.943} C_VEL
LIN {X 0,Y 417.36,Z 275.731,A -85,B 0,C 180,E1 20369.099,E2 20369.099} C_VEL
LIN {X 0,Y 417.332,Z 275.747,A -85,B 0,C 180,E1 20365.395,E2 20365.395} C_VEL
LIN {X 0,Y 417.315,Z 275.751,A -85,B 0,C 180,E1 20361.628,E2 20361.628} C_VEL
LIN {X 0,Y 417.308,Z 275.751,A -85,B 0,C 180,E1 20357.859,E2 20357.859} C_VEL
LIN {X 0,Y 417.308,Z 275.752,A -85,B 0,C 180,E1 20353.989,E2 20353.989} C_VEL
LIN {X 0,Y 417.324,Z 275.746,A -85,B 0,C 180,E1 20350.212,E2 20350.212} C_VEL
LIN {X 0,Y 417.353,Z 275.735,A -85,B 0,C 180,E1 20346.465,E2 20346.465} C_VEL
LIN {X 0,Y 417.362,Z 275.731,A -85,B 0,C 180,E1 20342.609,E2 20342.609} C_VEL
LIN {X 0,Y 417.364,Z 275.73,A -85,B 0,C 180,E1 20338.764,E2 20338.764} C_VEL
LIN {X 0,Y 417.353,Z 275.735,A -85,B 0,C 180,E1 20334.914,E2 20334.914} C_VEL
LIN {X 0,Y 417.341,Z 275.746,A -85,B 0,C 180,E1 20331.18,E2 20331.18} C_VEL
LIN {X 0,Y 417.336,Z 275.75,A -85,B 0,C 180,E1 20327.407,E2 20327.407} C_VEL
LIN {X 0,Y 417.344,Z 275.748,A -85,B 0,C 180,E1 20323.578,E2 20323.578} C_VEL
LIN {X 0,Y 417.351,Z 275.747,A -85,B 0,C 180,E1 20319.673,E2 20319.673} C_VEL
LIN {X 0,Y 417.367,Z 275.746,A -85,B 0,C 180,E1 20315.883,E2 20315.883} C_VEL
LIN {X 0,Y 417.381,Z 275.745,A -85,B 0,C 180,E1 20311.996,E2 20311.996} C_VEL
LIN {X 0,Y 417.375,Z 275.691,A -85,B 0,C 180,E1 20308.195,E2 20308.195} C_VEL
LIN {X 0,Y 417.376,Z 275.715,A -85,B 0,C 180,E1 20304.3,E2 20304.3} C_VEL
LIN {X 0,Y 417.388,Z 275.793,A -85,B 0,C 180,E1 20300.416,E2 20300.416} C_VEL
LIN {X 0,Y 417.49,Z 276.399,A -85,B 0,C 180,E1 20300.07,E2 20300.07} C_VEL
LIN {X 0,Y 419.009,Z 279.686,A -85,B 0,C 180,E1 20299.349,E2 20299.349} C_VEL
LIN {X 0,Y 424.057,Z 289.852,A -85,B 0,C 180,E1 20297.23,E2 20297.23} C_VEL
LIN {X 0,Y 431.015,Z 304.881,A -85,B 0,C 180,E1 20294.398,E2 20294.398} C_VEL
LIN {X 0,Y 438.144,Z 322,A -85,B 0,C 180,E1 20291.538,E2 20291.538} C_VEL
LIN {X 0,Y 439.835,Z 325.908,A -85,B 0,C 180,E1 20290.999,E2 20290.999} C_VEL
LIN {X 0,Y 444.608,Z 334.386,A -85,B 0,C 180,E1 20290.24,E2 20290.24} C_VEL
LIN {X 0,Y 449.133,Z 363.266,A -85,B 0,C 180,E1 20289.122,E2 20289.122} C_VEL
LIN {X 0,Y 443.581,Z 594.524,A -85,B 0,C 180,E1 20285.237,E2 20285.237} C_VEL
LIN {X 0,Y 442.379,Z 614.806,A -85,B 0,C 180,E1 20284.675,E2 20284.675} C_VEL
LIN {X 0,Y 440.796,Z 633.461,A -85,B 0,C 180,E1 20283.953,E2 20283.953} C_VEL
LIN {X 0,Y 439.234,Z 640.947,A -85,B 0,C 180,E1 20283.687,E2 20283.687} C_VEL
LIN {X 0,Y 432.206,Z 659.277,A -85,B 0,C 180,E1 20283.137,E2 20283.137} C_VEL
LIN {X 0,Y 430.464,Z 666.153,A -85,B 0,C 180,E1 20282.76,E2 20282.76} C_VEL
LIN {X 0,Y 427.832,Z 684.074,A -85,B 0,C 180,E1 20281.409,E2 20281.409} C_VEL
LIN {X 0,Y 424.994,Z 701.253,A -85,B 0,C 180,E1 20279.839,E2 20279.839} C_VEL
LIN {X 0,Y 421.977,Z 718.025,A -85,B 0,C 180,E1 20277.979,E2 20277.979} C_VEL
LIN {X 0,Y 419.09,Z 733.175,A -85,B 0,C 180,E1 20275.962,E2 20275.962} C_VEL
LIN {X 0,Y 416.466,Z 746.908,A -85,B 0,C 180,E1 20273.786,E2 20273.786} C_VEL
LIN {X 0,Y 414.067,Z 759.647,A -85,B 0,C 180,E1 20271.384,E2 20271.384} C_VEL
LIN {X 0,Y 412.066,Z 770.942,A -85,B 0,C 180,E1 20268.827,E2 20268.827} C_VEL
LIN {X 0,Y 410.484,Z 780.762,A -85,B 0,C 180,E1 20266.121,E2 20266.121} C_VEL
LIN {X 0,Y 409.332,Z 789.057,A -85,B 0,C 180,E1 20263.274,E2 20263.274} C_VEL
LIN {X 0,Y 408.623,Z 795.53,A -85,B 0,C 180,E1 20260.432,E2 20260.432} C_VEL
LIN {X 0,Y 408.226,Z 800.544,A -85,B 0,C 180,E1 20257.458,E2 20257.458} C_VEL
LIN {X 0,Y 408.062,Z 803.752,A -85,B 0,C 180,E1 20254.638,E2 20254.638} C_VEL
LIN {X 0,Y 408.006,Z 805.449,A -85,B 0,C 180,E1 20251.826,E2 20251.826} C_VEL
LIN {X 0,Y 407.999,Z 805.657,A -85,B 0,C 180,E1 20249.017,E2 20249.017} C_VEL
LIN {X 0,Y 408.036,Z 804.357,A -85,B 0,C 180,E1 20246.066,E2 20246.066} C_VEL
LIN {X 0,Y 408.168,Z 801.645,A -85,B 0,C 180,E1 20243.248,E2 20243.248} C_VEL
LIN {X 0,Y 408.493,Z 797.096,A -85,B 0,C 180,E1 20240.277,E2 20240.277} C_VEL
LIN {X 0,Y 409.094,Z 791.054,A -85,B 0,C 180,E1 20237.437,E2 20237.437} C_VEL
LIN {X 0,Y 410.104,Z 783.251,A -85,B 0,C 180,E1 20234.589,E2 20234.589} C_VEL
LIN {X 0,Y 411.623,Z 773.473,A -85,B 0,C 180,E1 20231.739,E2 20231.739} C_VEL
LIN {X 0,Y 413.501,Z 762.75,A -85,B 0,C 180,E1 20229.18,E2 20229.18} C_VEL
LIN {X 0,Y 415.848,Z 750.273,A -85,B 0,C 180,E1 20226.705,E2 20226.705} C_VEL
LIN {X 0,Y 418.552,Z 736.183,A -85,B 0,C 180,E1 20224.382,E2 20224.382} C_VEL
LIN {X 0,Y 421.329,Z 721.469,A -85,B 0,C 180,E1 20222.359,E2 20222.359} C_VEL
LIN {X 0,Y 424.267,Z 705.296,A -85,B 0,C 180,E1 20220.493,E2 20220.493} C_VEL
LIN {X 0,Y 427.299,Z 687.408,A -85,B 0,C 180,E1 20218.783,E2 20218.783} C_VEL
LIN {X 0,Y 429.932,Z 670.252,A -85,B 0,C 180,E1 20217.428,E2 20217.428} C_VEL
LIN {X 0,Y 432.443,Z 651.32,A -85,B 0,C 180,E1 20216.217,E2 20216.217} C_VEL
LIN {X 0,Y 434.475,Z 632.614,A -85,B 0,C 180,E1 20215.281,E2 20215.281} C_VEL
LIN {X 0,Y 436.223,Z 612.023,A -85,B 0,C 180,E1 20214.502,E2 20214.502} C_VEL
LIN {X 0,Y 437.392,Z 591.49,A -85,B 0,C 180,E1 20213.966,E2 20213.966} C_VEL
LIN {X 0,Y 443.15,Z 363.519,A -85,B 0,C 180,E1 20210.091,E2 20210.091} C_VEL
LIN {X 0,Y 438.84,Z 337.569,A -85,B 0,C 180,E1 20209.026,E2 20209.026} C_VEL
LIN {X 0,Y 431.082,Z 324.339,A -85,B 0,C 180,E1 20207.723,E2 20207.723} C_VEL
LIN {X 0,Y 424.021,Z 307.59,A -85,B 0,C 180,E1 20204.834,E2 20204.834} C_VEL
LIN {X 0,Y 417.38,Z 293.285,A -85,B 0,C 180,E1 20202.046,E2 20202.046} C_VEL
LIN {X 0,Y 413.208,Z 284.897,A -85,B 0,C 180,E1 20200.246,E2 20200.246} C_VEL
LIN {X 0,Y 410.943,Z 280.475,A -85,B 0,C 180,E1 20199.243,E2 20199.243} C_VEL
LIN {X 0,Y 409.463,Z 276.928,A -85,B 0,C 180,E1 20198.388,E2 20198.388} C_VEL
LIN {X 0,Y 409.428,Z 276.732,A -85,B 0,C 180,E1 20194.681,E2 20194.681} C_VEL
LIN {X 0,Y 409.418,Z 276.68,A -85,B 0,C 180,E1 20190.691,E2 20190.691} C_VEL
LIN {X 0,Y 409.423,Z 276.725,A -85,B 0,C 180,E1 20186.859,E2 20186.859} C_VEL
LIN {X 0,Y 409.424,Z 276.722,A -85,B 0,C 180,E1 20182.979,E2 20182.979} C_VEL
LIN {X 0,Y 409.426,Z 276.721,A -85,B 0,C 180,E1 20179.08,E2 20179.08} C_VEL
LIN {X 0,Y 409.431,Z 276.72,A -85,B 0,C 180,E1 20175.148,E2 20175.148} C_VEL
LIN {X 0,Y 409.434,Z 276.722,A -85,B 0,C 180,E1 20171.266,E2 20171.266} C_VEL
LIN {X 0,Y 409.44,Z 276.727,A -85,B 0,C 180,E1 20167.296,E2 20167.296} C_VEL
LIN {X 0,Y 409.432,Z 276.735,A -85,B 0,C 180,E1 20163.36,E2 20163.36} C_VEL
LIN {X 0,Y 409.439,Z 276.734,A -85,B 0,C 180,E1 20159.441,E2 20159.441} C_VEL
LIN {X 0,Y 409.418,Z 276.732,A -85,B 0,C 180,E1 20155.518,E2 20155.518} C_VEL
LIN {X 0,Y 409.397,Z 276.729,A -85,B 0,C 180,E1 20151.715,E2 20151.715} C_VEL
LIN {X 0,Y 409.378,Z 276.725,A -85,B 0,C 180,E1 20147.875,E2 20147.875} C_VEL
LIN {X 0,Y 409.362,Z 276.724,A -85,B 0,C 180,E1 20144.124,E2 20144.124} C_VEL
LIN {X 0,Y 409.37,Z 276.725,A -85,B 0,C 180,E1 20140.303,E2 20140.303} C_VEL
LIN {X 0,Y 409.384,Z 276.727,A -85,B 0,C 180,E1 20136.541,E2 20136.541} C_VEL
LIN {X 0,Y 409.405,Z 276.729,A -85,B 0,C 180,E1 20132.741,E2 20132.741} C_VEL
LIN {X 0,Y 409.427,Z 276.68,A -85,B 0,C 180,E1 20128.984,E2 20128.984} C_VEL
LIN {X 0,Y 409.439,Z 276.763,A -85,B 0,C 180,E1 20124.979,E2 20124.979} C_VEL
LIN {X 0,Y 409.499,Z 277.282,A -85,B 0,C 180,E1 20124.58,E2 20124.58} C_VEL
LIN {X 0,Y 410.902,Z 280.472,A -85,B 0,C 180,E1 20123.886,E2 20123.886} C_VEL
LIN {X 0,Y 412.233,Z 282.702,A -85,B 0,C 180,E1 20123.369,E2 20123.369} C_VEL
LIN {X 0,Y 417.123,Z 292.223,A -85,B 0,C 180,E1 20121.39,E2 20121.39} C_VEL
LIN {X 0,Y 422.919,Z 303.865,A -85,B 0,C 180,E1 20119.158,E2 20119.158} C_VEL
LIN {X 0,Y 424.91,Z 307.634,A -85,B 0,C 180,E1 20118.54,E2 20118.54} C_VEL
LIN {X 0,Y 437.673,Z 327.267,A -85,B 0,C 180,E1 20116.377,E2 20116.377} C_VEL
LIN {X 0,Y 446.618,Z 342.628,A -85,B 0,C 180,E1 20114.943,E2 20114.943} C_VEL
LIN {X 0,Y 439.729,Z 552.46,A -85,B 0,C 180,E1 20111.085,E2 20111.085} C_VEL
LIN {X 0,Y 437.831,Z 607.289,A -85,B 0,C 180,E1 20110.041,E2 20110.041} C_VEL
LIN {X 0,Y 436.214,Z 629.437,A -85,B 0,C 180,E1 20109.402,E2 20109.402} C_VEL
LIN {X 0,Y 434.228,Z 650.557,A -85,B 0,C 180,E1 20108.561,E2 20108.561} C_VEL
LIN {X 0,Y 431.902,Z 671.271,A -85,B 0,C 180,E1 20107.505,E2 20107.505} C_VEL
LIN {X 0,Y 429.233,Z 691.872,A -85,B 0,C 180,E1 20106.192,E2 20106.192} C_VEL
LIN {X 0,Y 426.384,Z 711.572,A -85,B 0,C 180,E1 20104.655,E2 20104.655} C_VEL
LIN {X 0,Y 423.354,Z 731.258,A -85,B 0,C 180,E1 20102.82,E2 20102.82} C_VEL
LIN {X 0,Y 420.495,Z 749.333,A -85,B 0,C 180,E1 20100.824,E2 20100.824} C_VEL
LIN {X 0,Y 417.73,Z 766.44,A -85,B 0,C 180,E1 20098.6,E2 20098.6} C_VEL
LIN {X 0,Y 415.333,Z 781.572,A -85,B 0,C 180,E1 20096.292,E2 20096.292} C_VEL
LIN {X 0,Y 413.141,Z 796.223,A -85,B 0,C 180,E1 20093.686,E2 20093.686} C_VEL
LIN {X 0,Y 411.414,Z 808.789,A -85,B 0,C 180,E1 20091.056,E2 20091.056} C_VEL
LIN {X 0,Y 410.068,Z 819.639,A -85,B 0,C 180,E1 20088.332,E2 20088.332} C_VEL
LIN {X 0,Y 409.082,Z 829.168,A -85,B 0,C 180,E1 20085.45,E2 20085.45} C_VEL
LIN {X 0,Y 408.457,Z 836.891,A -85,B 0,C 180,E1 20082.583,E2 20082.583} C_VEL
LIN {X 0,Y 408.125,Z 842.797,A -85,B 0,C 180,E1 20079.732,E2 20079.732} C_VEL
LIN {X 0,Y 407.975,Z 847.332,A -85,B 0,C 180,E1 20076.756,E2 20076.756} C_VEL
LIN {X 0,Y 407.932,Z 850.015,A -85,B 0,C 180,E1 20074.076,E2 20074.076} C_VEL
LIN {X 0,Y 407.933,Z 851.401,A -85,B 0,C 180,E1 20071.124,E2 20071.124} C_VEL
LIN {X 0,Y 407.925,Z 851.328,A -85,B 0,C 180,E1 20068.455,E2 20068.455} C_VEL
LIN {X 0,Y 407.939,Z 849.658,A -85,B 0,C 180,E1 20065.502,E2 20065.502} C_VEL
LIN {X 0,Y 407.995,Z 846.656,A -85,B 0,C 180,E1 20062.679,E2 20062.679} C_VEL
LIN {X 0,Y 408.159,Z 842,A -85,B 0,C 180,E1 20059.841,E2 20059.841} C_VEL
LIN {X 0,Y 408.557,Z 835.469,A -85,B 0,C 180,E1 20056.845,E2 20056.845} C_VEL
LIN {X 0,Y 409.242,Z 827.465,A -85,B 0,C 180,E1 20053.974,E2 20053.974} C_VEL
LIN {X 0,Y 410.248,Z 818.029,A -85,B 0,C 180,E1 20051.234,E2 20051.234} C_VEL
LIN {X 0,Y 411.7,Z 806.612,A -85,B 0,C 180,E1 20048.459,E2 20048.459} C_VEL
LIN {X 0,Y 413.482,Z 794.012,A -85,B 0,C 180,E1 20045.88,E2 20045.88} C_VEL
LIN {X 0,Y 415.612,Z 779.791,A -85,B 0,C 180,E1 20043.419,E2 20043.419} C_VEL
LIN {X 0,Y 418.218,Z 763.265,A -85,B 0,C 180,E1 20040.967,E2 20040.967} C_VEL
LIN {X 0,Y 420.977,Z 746.317,A -85,B 0,C 180,E1 20038.818,E2 20038.818} C_VEL
LIN {X 0,Y 423.86,Z 728.205,A -85,B 0,C 180,E1 20036.868,E2 20036.868} C_VEL
LIN {X 0,Y 426.749,Z 709.062,A -85,B 0,C 180,E1 20035.133,E2 20035.133} C_VEL
LIN {X 0,Y 429.717,Z 688.098,A -85,B 0,C 180,E1 20033.553,E2 20033.553} C_VEL
LIN {X 0,Y 432.358,Z 667.587,A -85,B 0,C 180,E1 20032.29,E2 20032.29} C_VEL
LIN {X 0,Y 434.547,Z 647.452,A -85,B 0,C 180,E1 20031.299,E2 20031.299} C_VEL
LIN {X 0,Y 436.501,Z 625.542,A -85,B 0,C 180,E1 20030.472,E2 20030.472} C_VEL
LIN {X 0,Y 438.045,Z 602.78,A -85,B 0,C 180,E1 20029.865,E2 20029.865} C_VEL
LIN {X 0,Y 444.965,Z 392.608,A -85,B 0,C 180,E1 20025.975,E2 20025.975} C_VEL
LIN {X 0,Y 446.516,Z 342.285,A -85,B 0,C 180,E1 20025.04,E2 20025.04} C_VEL
LIN {X 0,Y 434.279,Z 321.944,A -85,B 0,C 180,E1 20023.073,E2 20023.073} C_VEL
LIN {X 0,Y 424.163,Z 306.39,A -85,B 0,C 180,E1 20021.302,E2 20021.302} C_VEL
LIN {X 0,Y 418.035,Z 293.983,A -85,B 0,C 180,E1 20018.979,E2 20018.979} C_VEL
LIN {X 0,Y 413.537,Z 285.26,A -85,B 0,C 180,E1 20017.189,E2 20017.189} C_VEL
LIN {X 0,Y 411.569,Z 281.281,A -85,B 0,C 180,E1 20016.353,E2 20016.353} C_VEL
LIN {X 0,Y 409.782,Z 278.351,A -85,B 0,C 180,E1 20015.66,E2 20015.66} C_VEL
LIN {X 0,Y 409.444,Z 276.933,A -85,B 0,C 180,E1 20015.313,E2 20015.313} C_VEL
LIN {X 0,Y 409.392,Z 276.684,A -85,B 0,C 180,E1 20011.51,E2 20011.51} C_VEL
LIN {X 0,Y 409.385,Z 276.74,A -85,B 0,C 180,E1 20007.806,E2 20007.806} C_VEL
LIN {X 0,Y 409.378,Z 276.732,A -85,B 0,C 180,E1 20003.918,E2 20003.918} C_VEL
LIN {X 0,Y 409.381,Z 276.727,A -85,B 0,C 180,E1 20000.143,E2 20000.143} C_VEL
LIN {X 0,Y 409.385,Z 276.725,A -85,B 0,C 180,E1 19996.312,E2 19996.312} C_VEL
LIN {X 0,Y 409.405,Z 276.727,A -85,B 0,C 180,E1 19992.554,E2 19992.554} C_VEL
LIN {X 0,Y 409.417,Z 276.73,A -85,B 0,C 180,E1 19988.567,E2 19988.567} C_VEL
LIN {X 0,Y 409.422,Z 276.734,A -85,B 0,C 180,E1 19984.622,E2 19984.622} C_VEL
LIN {X 0,Y 409.433,Z 276.738,A -85,B 0,C 180,E1 19980.699,E2 19980.699} C_VEL
LIN {X 0,Y 409.422,Z 276.733,A -85,B 0,C 180,E1 19976.78,E2 19976.78} C_VEL
LIN {X 0,Y 409.423,Z 276.726,A -85,B 0,C 180,E1 19972.845,E2 19972.845} C_VEL
LIN {X 0,Y 409.409,Z 276.721,A -85,B 0,C 180,E1 19969.018,E2 19969.018} C_VEL
LIN {X 0,Y 409.401,Z 276.72,A -85,B 0,C 180,E1 19965.263,E2 19965.263} C_VEL
LIN {X 0,Y 409.406,Z 276.721,A -85,B 0,C 180,E1 19961.341,E2 19961.341} C_VEL
LIN {X 0,Y 409.41,Z 276.721,A -85,B 0,C 180,E1 19957.387,E2 19957.387} C_VEL
LIN {X 0,Y 409.416,Z 276.722,A -85,B 0,C 180,E1 19953.454,E2 19953.454} C_VEL
LIN {X 0,Y 409.416,Z 276.684,A -85,B 0,C 180,E1 19949.548,E2 19949.548} C_VEL
LIN {X 0,Y 409.43,Z 276.738,A -85,B 0,C 180,E1 19945.629,E2 19945.629} C_VEL
LIN {X 0,Y 409.443,Z 276.793,A -85,B 0,C 180,E1 19941.664,E2 19941.664} C_VEL
LIN {X 0,Y 409.578,Z 277.555,A -85,B 0,C 180,E1 19941.322,E2 19941.322} C_VEL
LIN {X 0,Y 411.466,Z 281.164,A -85,B 0,C 180,E1 19940.457,E2 19940.457} C_VEL
LIN {X 0,Y 418.047,Z 294.473,A -85,B 0,C 180,E1 19937.587,E2 19937.587} C_VEL
LIN {X 0,Y 425.227,Z 310.338,A -85,B 0,C 180,E1 19934.564,E2 19934.564} C_VEL
LIN {X 0,Y 431.462,Z 325.112,A -85,B 0,C 180,E1 19932.086,E2 19932.086} C_VEL
LIN {X 0,Y 439.096,Z 338.281,A -85,B 0,C 180,E1 19930.827,E2 19930.827} C_VEL
LIN {X 0,Y 443.131,Z 364.809,A -85,B 0,C 180,E1 19929.785,E2 19929.785} C_VEL
LIN {X 0,Y 437.266,Z 594.598,A -85,B 0,C 180,E1 19925.879,E2 19925.879} C_VEL
LIN {X 0,Y 436.007,Z 614.94,A -85,B 0,C 180,E1 19925.311,E2 19925.311} C_VEL
LIN {X 0,Y 434.238,Z 634.712,A -85,B 0,C 180,E1 19924.532,E2 19924.532} C_VEL
LIN {X 0,Y 432.02,Z 654.455,A -85,B 0,C 180,E1 19923.502,E2 19923.502} C_VEL
LIN {X 0,Y 430.464,Z 666.153,A -85,B 0,C 180,E1 19922.76,E2 19922.76} C_VEL
LIN {X 0,Y 428.659,Z 673.155,A -85,B 0,C 180,E1 19922.348,E2 19922.348} C_VEL
LIN {X 0,Y 420.914,Z 690.387,A -85,B 0,C 180,E1 19921.417,E2 19921.417} C_VEL
LIN {X 0,Y 418.969,Z 696.732,A -85,B 0,C 180,E1 19920.896,E2 19920.896} C_VEL
LIN {X 0,Y 415.777,Z 713.949,A -85,B 0,C 180,E1 19919.062,E2 19919.062} C_VEL
LIN {X 0,Y 412.762,Z 729.37,A -85,B 0,C 180,E1 19917.09,E2 19917.09} C_VEL
LIN {X 0,Y 409.929,Z 743.369,A -85,B 0,C 180,E1 19914.958,E2 19914.958} C_VEL
LIN {X 0,Y 407.23,Z 756.702,A -85,B 0,C 180,E1 19912.52,E2 19912.52} C_VEL
LIN {X 0,Y 405.052,Z 767.908,A -85,B 0,C 180,E1 19910.066,E2 19910.066} C_VEL
LIN {X 0,Y 403.165,Z 778.419,A -85,B 0,C 180,E1 19907.29,E2 19907.29} C_VEL
LIN {X 0,Y 401.848,Z 786.87,A -85,B 0,C 180,E1 19904.554,E2 19904.554} C_VEL
LIN {X 0,Y 400.924,Z 794.001,A -85,B 0,C 180,E1 19901.654,E2 19901.654} C_VEL
LIN {X 0,Y 400.386,Z 799.568,A -85,B 0,C 180,E1 19898.617,E2 19898.617} C_VEL
LIN {X 0,Y 400.122,Z 803.242,A -85,B 0,C 180,E1 19895.736,E2 19895.736} C_VEL
LIN {X 0,Y 400.028,Z 805.517,A -85,B 0,C 180,E1 19892.722,E2 19892.722} C_VEL
LIN {X 0,Y 400.014,Z 806.233,A -85,B 0,C 180,E1 19889.857,E2 19889.857} C_VEL
LIN {X 0,Y 400.029,Z 805.433,A -85,B 0,C 180,E1 19886.991,E2 19886.991} C_VEL
LIN {X 0,Y 400.136,Z 803.07,A -85,B 0,C 180,E1 19884.003,E2 19884.003} C_VEL
LIN {X 0,Y 400.429,Z 799.004,A -85,B 0,C 180,E1 19880.95,E2 19880.95} C_VEL
LIN {X 0,Y 400.972,Z 793.546,A -85,B 0,C 180,E1 19878.056,E2 19878.056} C_VEL
LIN {X 0,Y 401.934,Z 786.346,A -85,B 0,C 180,E1 19875.154,E2 19875.154} C_VEL
LIN {X 0,Y 403.3,Z 777.669,A -85,B 0,C 180,E1 19872.395,E2 19872.395} C_VEL
LIN {X 0,Y 405.196,Z 767.178,A -85,B 0,C 180,E1 19869.667,E2 19869.667} C_VEL
LIN {X 0,Y 407.582,Z 754.936,A -85,B 0,C 180,E1 19867.043,E2 19867.043} C_VEL
LIN {X 0,Y 410.201,Z 742.006,A -85,B 0,C 180,E1 19864.731,E2 19864.731} C_VEL
LIN {X 0,Y 413.165,Z 727.467,A -85,B 0,C 180,E1 19862.549,E2 19862.549} C_VEL
LIN {X 0,Y 416.272,Z 711.56,A -85,B 0,C 180,E1 19860.563,E2 19860.563} C_VEL
LIN {X 0,Y 419.298,Z 694.956,A -85,B 0,C 180,E1 19858.839,E2 19858.839} C_VEL
LIN {X 0,Y 422.244,Z 677.354,A -85,B 0,C 180,E1 19857.325,E2 19857.325} C_VEL
LIN {X 0,Y 424.975,Z 658.933,A -85,B 0,C 180,E1 19856.03,E2 19856.03} C_VEL
LIN {X 0,Y 427.354,Z 639.772,A -85,B 0,C 180,E1 19854.953,E2 19854.953} C_VEL
LIN {X 0,Y 429.365,Z 619.309,A -85,B 0,C 180,E1 19854.087,E2 19854.087} C_VEL
LIN {X 0,Y 430.759,Z 599.295,A -85,B 0,C 180,E1 19853.482,E2 19853.482} C_VEL
LIN {X 0,Y 431.743,Z 571.759,A -85,B 0,C 180,E1 19852.95,E2 19852.95} C_VEL
LIN {X 0,Y 437.196,Z 364.824,A -85,B 0,C 180,E1 19849.401,E2 19849.401} C_VEL
LIN {X 0,Y 433.384,Z 341.538,A -85,B 0,C 180,E1 19848.424,E2 19848.424} C_VEL
LIN {X 0,Y 422.771,Z 323.674,A -85,B 0,C 180,E1 19846.557,E2 19846.557} C_VEL
LIN {X 0,Y 415.894,Z 307.599,A -85,B 0,C 180,E1 19843.629,E2 19843.629} C_VEL
LIN {X 0,Y 409.874,Z 294.854,A -85,B 0,C 180,E1 19841.012,E2 19841.012} C_VEL
LIN {X 0,Y 405.328,Z 285.922,A -85,B 0,C 180,E1 19838.979,E2 19838.979} C_VEL
LIN {X 0,Y 403.152,Z 281.637,A -85,B 0,C 180,E1 19837.957,E2 19837.957} C_VEL
LIN {X 0,Y 401.524,Z 277.926,A -85,B 0,C 180,E1 19837.01,E2 19837.01} C_VEL
LIN {X 0,Y 401.495,Z 277.693,A -85,B 0,C 180,E1 19833.203,E2 19833.203} C_VEL
LIN {X 0,Y 401.499,Z 277.693,A -85,B 0,C 180,E1 19829.216,E2 19829.216} C_VEL
LIN {X 0,Y 401.495,Z 277.714,A -85,B 0,C 180,E1 19825.205,E2 19825.205} C_VEL
LIN {X 0,Y 401.502,Z 277.714,A -85,B 0,C 180,E1 19821.321,E2 19821.321} C_VEL
LIN {X 0,Y 401.501,Z 277.714,A -85,B 0,C 180,E1 19817.388,E2 19817.388} C_VEL
LIN {X 0,Y 401.503,Z 277.711,A -85,B 0,C 180,E1 19813.391,E2 19813.391} C_VEL
LIN {X 0,Y 401.498,Z 277.706,A -85,B 0,C 180,E1 19809.46,E2 19809.46} C_VEL
LIN {X 0,Y 401.491,Z 277.704,A -85,B 0,C 180,E1 19805.574,E2 19805.574} C_VEL
LIN {X 0,Y 401.486,Z 277.706,A -85,B 0,C 180,E1 19801.57,E2 19801.57} C_VEL
LIN {X 0,Y 401.468,Z 277.711,A -85,B 0,C 180,E1 19797.717,E2 19797.717} C_VEL
LIN {X 0,Y 401.454,Z 277.719,A -85,B 0,C 180,E1 19793.852,E2 19793.852} C_VEL
LIN {X 0,Y 401.436,Z 277.729,A -85,B 0,C 180,E1 19790.104,E2 19790.104} C_VEL
LIN {X 0,Y 401.428,Z 277.73,A -85,B 0,C 180,E1 19786.166,E2 19786.166} C_VEL
LIN {X 0,Y 401.429,Z 277.729,A -85,B 0,C 180,E1 19782.16,E2 19782.16} C_VEL
LIN {X 0,Y 401.435,Z 277.728,A -85,B 0,C 180,E1 19778.216,E2 19778.216} C_VEL
LIN {X 0,Y 401.443,Z 277.722,A -85,B 0,C 180,E1 19774.318,E2 19774.318} C_VEL
LIN {X 0,Y 401.45,Z 277.694,A -85,B 0,C 180,E1 19770.453,E2 19770.453} C_VEL
LIN {X 0,Y 401.465,Z 277.703,A -85,B 0,C 180,E1 19766.605,E2 19766.605} C_VEL
LIN {X 0,Y 401.544,Z 278.293,A -85,B 0,C 180,E1 19765.975,E2 19765.975} C_VEL
LIN {X 0,Y 403.145,Z 281.667,A -85,B 0,C 180,E1 19765.176,E2 19765.176} C_VEL
LIN {X 0,Y 404.283,Z 283.641,A -85,B 0,C 180,E1 19764.698,E2 19764.698} C_VEL
LIN {X 0,Y 407.022,Z 288.839,A -85,B 0,C 180,E1 19763.525,E2 19763.525} C_VEL
LIN {X 0,Y 413.203,Z 300.743,A -85,B 0,C 180,E1 19761.014,E2 19761.014} C_VEL
LIN {X 0,Y 416.581,Z 307.595,A -85,B 0,C 180,E1 19759.746,E2 19759.746} C_VEL
LIN {X 0,Y 428.463,Z 325.513,A -85,B 0,C 180,E1 19757.615,E2 19757.615} C_VEL
LIN {X 0,Y 440.068,Z 344.687,A -85,B 0,C 180,E1 19755.681,E2 19755.681} C_VEL
LIN {X 0,Y 440.61,Z 346.1,A -85,B 0,C 180,E1 19755.583,E2 19755.583} C_VEL
LIN {X 0,Y 433.406,Z 554.958,A -85,B 0,C 180,E1 19751.699,E2 19751.699} C_VEL
LIN {X 0,Y 431.501,Z 607.143,A -85,B 0,C 180,E1 19750.691,E2 19750.691} C_VEL
LIN {X 0,Y 429.801,Z 629.373,A -85,B 0,C 180,E1 19750.043,E2 19750.043} C_VEL
LIN {X 0,Y 427.693,Z 650.731,A -85,B 0,C 180,E1 19749.181,E2 19749.181} C_VEL
LIN {X 0,Y 425.252,Z 671.394,A -85,B 0,C 180,E1 19748.11,E2 19748.11} C_VEL
LIN {X 0,Y 422.448,Z 691.928,A -85,B 0,C 180,E1 19746.783,E2 19746.783} C_VEL
LIN {X 0,Y 419.453,Z 711.537,A -85,B 0,C 180,E1 19745.229,E2 19745.229} C_VEL
LIN {X 0,Y 416.264,Z 731.142,A -85,B 0,C 180,E1 19743.37,E2 19743.37} C_VEL
LIN {X 0,Y 413.242,Z 749.143,A -85,B 0,C 180,E1 19741.345,E2 19741.345} C_VEL
LIN {X 0,Y 410.312,Z 766.185,A -85,B 0,C 180,E1 19739.087,E2 19739.087} C_VEL
LIN {X 0,Y 407.701,Z 781.65,A -85,B 0,C 180,E1 19736.666,E2 19736.666} C_VEL
LIN {X 0,Y 405.388,Z 796.137,A -85,B 0,C 180,E1 19734.013,E2 19734.013} C_VEL
LIN {X 0,Y 403.561,Z 808.696,A -85,B 0,C 180,E1 19731.319,E2 19731.319} C_VEL
LIN {X 0,Y 402.217,Z 818.95,A -85,B 0,C 180,E1 19728.703,E2 19728.703} C_VEL
LIN {X 0,Y 401.162,Z 828.544,A -85,B 0,C 180,E1 19725.763,E2 19725.763} C_VEL
LIN {X 0,Y 400.522,Z 836.003,A -85,B 0,C 180,E1 19722.983,E2 19722.983} C_VEL
LIN {X 0,Y 400.152,Z 842.015,A -85,B 0,C 180,E1 19720.073,E2 19720.073} C_VEL
LIN {X 0,Y 399.996,Z 846.692,A -85,B 0,C 180,E1 19717.035,E2 19717.035} C_VEL
LIN {X 0,Y 399.945,Z 849.438,A -85,B 0,C 180,E1 19714.301,E2 19714.301} C_VEL
LIN {X 0,Y 399.942,Z 850.928,A -85,B 0,C 180,E1 19711.289,E2 19711.289} C_VEL
LIN {X 0,Y 399.939,Z 850.903,A -85,B 0,C 180,E1 19708.567,E2 19708.567} C_VEL
LIN {X 0,Y 399.948,Z 849.315,A -85,B 0,C 180,E1 19705.555,E2 19705.555} C_VEL
LIN {X 0,Y 400.001,Z 846.351,A -85,B 0,C 180,E1 19702.676,E2 19702.676} C_VEL
LIN {X 0,Y 400.166,Z 841.754,A -85,B 0,C 180,E1 19699.782,E2 19699.782} C_VEL
LIN {X 0,Y 400.566,Z 835.394,A -85,B 0,C 180,E1 19696.775,E2 19696.775} C_VEL
LIN {X 0,Y 401.246,Z 827.701,A -85,B 0,C 180,E1 19693.943,E2 19693.943} C_VEL
LIN {X 0,Y 402.345,Z 817.874,A -85,B 0,C 180,E1 19691.002,E2 19691.002} C_VEL
LIN {X 0,Y 403.859,Z 806.564,A -85,B 0,C 180,E1 19688.188,E2 19688.188} C_VEL
LIN {X 0,Y 405.741,Z 793.924,A -85,B 0,C 180,E1 19685.544,E2 19685.544} C_VEL
LIN {X 0,Y 407.994,Z 779.88,A -85,B 0,C 180,E1 19683.04,E2 19683.04} C_VEL
LIN {X 0,Y 410.749,Z 763.545,A -85,B 0,C 180,E1 19680.548,E2 19680.548} C_VEL
LIN {X 0,Y 413.649,Z 746.777,A -85,B 0,C 180,E1 19678.365,E2 19678.365} C_VEL
LIN {X 0,Y 416.748,Z 728.374,A -85,B 0,C 180,E1 19676.345,E2 19676.345} C_VEL
LIN {X 0,Y 419.8,Z 709.251,A -85,B 0,C 180,E1 19674.577,E2 19674.577} C_VEL
LIN {X 0,Y 422.864,Z 688.825,A -85,B 0,C 180,E1 19673.005,E2 19673.005} C_VEL
LIN {X 0,Y 425.575,Z 669.044,A -85,B 0,C 180,E1 19671.753,E2 19671.753} C_VEL
LIN {X 0,Y 427.932,Z 648.448,A -85,B 0,C 180,E1 19670.716,E2 19670.716} C_VEL
LIN {X 0,Y 430.059,Z 625.992,A -85,B 0,C 180,E1 19669.847,E2 19669.847} C_VEL
LIN {X 0,Y 431.674,Z 603.635,A -85,B 0,C 180,E1 19669.235,E2 19669.235} C_VEL
LIN {X 0,Y 438.823,Z 397.477,A -85,B 0,C 180,E1 19665.372,E2 19665.372} C_VEL
LIN {X 0,Y 440.458,Z 345.369,A -85,B 0,C 180,E1 19664.385,E2 19664.385} C_VEL
LIN {X 0,Y 428.896,Z 326.241,A -85,B 0,C 180,E1 19662.468,E2 19662.468} C_VEL
LIN {X 0,Y 416.825,Z 307.964,A -85,B 0,C 180,E1 19660.32,E2 19660.32} C_VEL
LIN {X 0,Y 413.819,Z 302.216,A -85,B 0,C 180,E1 19659.274,E2 19659.274} C_VEL
LIN {X 0,Y 408.36,Z 291.261,A -85,B 0,C 180,E1 19657.036,E2 19657.036} C_VEL
LIN {X 0,Y 405.634,Z 286.305,A -85,B 0,C 180,E1 19655.919,E2 19655.919} C_VEL
LIN {X 0,Y 403.38,Z 281.959,A -85,B 0,C 180,E1 19654.93,E2 19654.93} C_VEL
LIN {X 0,Y 401.566,Z 278.394,A -85,B 0,C 180,E1 19654.071,E2 19654.071} C_VEL
LIN {X 0,Y 401.462,Z 277.772,A -85,B 0,C 180,E1 19653.714,E2 19653.714} C_VEL
LIN {X 0,Y 401.443,Z 277.687,A -85,B 0,C 180,E1 19649.876,E2 19649.876} C_VEL
LIN {X 0,Y 401.443,Z 277.718,A -85,B 0,C 180,E1 19645.96,E2 19645.96} C_VEL
LIN {X 0,Y 401.443,Z 277.721,A -85,B 0,C 180,E1 19642.091,E2 19642.091} C_VEL
LIN {X 0,Y 401.448,Z 277.72,A -85,B 0,C 180,E1 19638.289,E2 19638.289} C_VEL
LIN {X 0,Y 401.455,Z 277.718,A -85,B 0,C 180,E1 19634.422,E2 19634.422} C_VEL
LIN {X 0,Y 401.463,Z 277.715,A -85,B 0,C 180,E1 19630.475,E2 19630.475} C_VEL
LIN {X 0,Y 401.484,Z 277.709,A -85,B 0,C 180,E1 19626.578,E2 19626.578} C_VEL
LIN {X 0,Y 401.481,Z 277.707,A -85,B 0,C 180,E1 19622.569,E2 19622.569} C_VEL
LIN {X 0,Y 401.488,Z 277.706,A -85,B 0,C 180,E1 19618.715,E2 19618.715} C_VEL
LIN {X 0,Y 401.488,Z 277.707,A -85,B 0,C 180,E1 19614.713,E2 19614.713} C_VEL
LIN {X 0,Y 401.474,Z 277.716,A -85,B 0,C 180,E1 19610.973,E2 19610.973} C_VEL
LIN {X 0,Y 401.472,Z 277.724,A -85,B 0,C 180,E1 19607.047,E2 19607.047} C_VEL
LIN {X 0,Y 401.471,Z 277.728,A -85,B 0,C 180,E1 19603.208,E2 19603.208} C_VEL
LIN {X 0,Y 401.473,Z 277.727,A -85,B 0,C 180,E1 19599.289,E2 19599.289} C_VEL
LIN {X 0,Y 401.476,Z 277.727,A -85,B 0,C 180,E1 19595.366,E2 19595.366} C_VEL
LIN {X 0,Y 401.479,Z 277.718,A -85,B 0,C 180,E1 19591.434,E2 19591.434} C_VEL
LIN {X 0,Y 401.478,Z 277.676,A -85,B 0,C 180,E1 19587.456,E2 19587.456} C_VEL
LIN {X 0,Y 401.484,Z 277.675,A -85,B 0,C 180,E1 19583.55,E2 19583.55} C_VEL
LIN {X 0,Y 401.577,Z 278.217,A -85,B 0,C 180,E1 19582.769,E2 19582.769} C_VEL
LIN {X 0,Y 403.283,Z 281.822,A -85,B 0,C 180,E1 19581.877,E2 19581.877} C_VEL
LIN {X 0,Y 406.716,Z 288.681,A -85,B 0,C 180,E1 19580.269,E2 19580.269} C_VEL
LIN {X 0,Y 410.966,Z 297.233,A -85,B 0,C 180,E1 19578.379,E2 19578.379} C_VEL
LIN {X 0,Y 417.404,Z 311.013,A -85,B 0,C 180,E1 19575.616,E2 19575.616} C_VEL
LIN {X 0,Y 423.295,Z 324.764,A -85,B 0,C 180,E1 19573.197,E2 19573.197} C_VEL
LIN {X 0,Y 433.629,Z 342.193,A -85,B 0,C 180,E1 19571.429,E2 19571.429} C_VEL
LIN {X 0,Y 437.196,Z 366.219,A -85,B 0,C 180,E1 19570.468,E2 19570.468} C_VEL
LIN {X 0,Y 430.997,Z 594.833,A -85,B 0,C 180,E1 19566.535,E2 19566.535} C_VEL
LIN {X 0,Y 429.68,Z 615.174,A -85,B 0,C 180,E1 19565.962,E2 19565.962} C_VEL
LIN {X 0,Y 427.818,Z 635.077,A -85,B 0,C 180,E1 19565.169,E2 19565.169} C_VEL
LIN {X 0,Y 425.414,Z 655.381,A -85,B 0,C 180,E1 19564.093,E2 19564.093} C_VEL
LIN {X 0,Y 422.819,Z 673.659,A -85,B 0,C 180,E1 19562.867,E2 19562.867} C_VEL
LIN {X 0,Y 419.967,Z 691.175,A -85,B 0,C 180,E1 19561.425,E2 19561.425} C_VEL
LIN {X 0,Y 418.969,Z 696.732,A -85,B 0,C 180,E1 19560.896,E2 19560.896} C_VEL
LIN {X 0,Y 416.993,Z 703.119,A -85,B 0,C 180,E1 19560.338,E2 19560.338} C_VEL
LIN {X 0,Y 408.804,Z 718.822,A -85,B 0,C 180,E1 19559.02,E2 19559.02} C_VEL
LIN {X 0,Y 406.727,Z 724.539,A -85,B 0,C 180,E1 19558.353,E2 19558.353} C_VEL
LIN {X 0,Y 403.561,Z 739.479,A -85,B 0,C 180,E1 19556.168,E2 19556.168} C_VEL
LIN {X 0,Y 400.715,Z 752.81,A -85,B 0,C 180,E1 19553.842,E2 19553.842} C_VEL
LIN {X 0,Y 398.179,Z 764.934,A -85,B 0,C 180,E1 19551.312,E2 19551.312} C_VEL
LIN {X 0,Y 396.024,Z 775.813,A -85,B 0,C 180,E1 19548.549,E2 19548.549} C_VEL
LIN {X 0,Y 394.416,Z 784.852,A -85,B 0,C 180,E1 19545.738,E2 19545.738} C_VEL
LIN {X 0,Y 393.27,Z 792.482,A -85,B 0,C 180,E1 19542.779,E2 19542.779} C_VEL
LIN {X 0,Y 392.565,Z 798.56,A -85,B 0,C 180,E1 19539.705,E2 19539.705} C_VEL
LIN {X 0,Y 392.22,Z 802.804,A -85,B 0,C 180,E1 19536.734,E2 19536.734} C_VEL
LIN {X 0,Y 392.062,Z 805.512,A -85,B 0,C 180,E1 19533.655,E2 19533.655} C_VEL
LIN {X 0,Y 392.024,Z 806.582,A -85,B 0,C 180,E1 19530.731,E2 19530.731} C_VEL
LIN {X 0,Y 392.033,Z 806.199,A -85,B 0,C 180,E1 19527.661,E2 19527.661} C_VEL
LIN {X 0,Y 392.121,Z 804.397,A -85,B 0,C 180,E1 19524.733,E2 19524.733} C_VEL
LIN {X 0,Y 392.37,Z 800.825,A -85,B 0,C 180,E1 19521.648,E2 19521.648} C_VEL
LIN {X 0,Y 392.865,Z 795.81,A -85,B 0,C 180,E1 19518.699,E2 19518.699} C_VEL
LIN {X 0,Y 393.802,Z 788.754,A -85,B 0,C 180,E1 19515.593,E2 19515.593} C_VEL
LIN {X 0,Y 395.227,Z 780.133,A -85,B 0,C 180,E1 19512.632,E2 19512.632} C_VEL
LIN {X 0,Y 397.074,Z 770.433,A -85,B 0,C 180,E1 19509.925,E2 19509.925} C_VEL
LIN {X 0,Y 399.385,Z 759.125,A -85,B 0,C 180,E1 19507.323,E2 19507.323} C_VEL
LIN {X 0,Y 401.979,Z 746.908,A -85,B 0,C 180,E1 19504.986,E2 19504.986} C_VEL
LIN {X 0,Y 405.057,Z 732.512,A -85,B 0,C 180,E1 19502.67,E2 19502.67} C_VEL
LIN {X 0,Y 408.286,Z 717.064,A -85,B 0,C 180,E1 19500.594,E2 19500.594} C_VEL
LIN {X 0,Y 411.477,Z 701.081,A -85,B 0,C 180,E1 19498.797,E2 19498.797} C_VEL
LIN {X 0,Y 414.697,Z 683.302,A -85,B 0,C 180,E1 19497.148,E2 19497.148} C_VEL
LIN {X 0,Y 417.622,Z 664.987,A -85,B 0,C 180,E1 19495.763,E2 19495.763} C_VEL
LIN {X 0,Y 420.265,Z 645.76,A -85,B 0,C 180,E1 19494.599,E2 19494.599} C_VEL
LIN {X 0,Y 422.449,Z 626.059,A -85,B 0,C 180,E1 19493.671,E2 19493.671} C_VEL
LIN {X 0,Y 424.164,Z 605.755,A -85,B 0,C 180,E1 19492.968,E2 19492.968} C_VEL
LIN {X 0,Y 425.242,Z 584.389,A -85,B 0,C 180,E1 19492.483,E2 19492.483} C_VEL
LIN {X 0,Y 431.347,Z 366.421,A -85,B 0,C 180,E1 19488.704,E2 19488.704} C_VEL
LIN {X 0,Y 428.044,Z 345.777,A -85,B 0,C 180,E1 19487.822,E2 19487.822} C_VEL
LIN {X 0,Y 417.326,Z 327.963,A -85,B 0,C 180,E1 19485.928,E2 19485.928} C_VEL
LIN {X 0,Y 414.562,Z 323.272,A -85,B 0,C 180,E1 19485.357,E2 19485.357} C_VEL
LIN {X 0,Y 407.996,Z 308.278,A -85,B 0,C 180,E1 19482.47,E2 19482.47} C_VEL
LIN {X 0,Y 402.3,Z 296.306,A -85,B 0,C 180,E1 19479.883,E2 19479.883} C_VEL
LIN {X 0,Y 397.569,Z 287.12,A -85,B 0,C 180,E1 19477.672,E2 19477.672} C_VEL
LIN {X 0,Y 395.486,Z 282.986,A -85,B 0,C 180,E1 19476.631,E2 19476.631} C_VEL
LIN {X 0,Y 393.748,Z 279.675,A -85,B 0,C 180,E1 19475.736,E2 19475.736} C_VEL
LIN {X 0,Y 393.57,Z 278.789,A -85,B 0,C 180,E1 19475.366,E2 19475.366} C_VEL
LIN {X 0,Y 393.559,Z 278.649,A -85,B 0,C 180,E1 19471.387,E2 19471.387} C_VEL
LIN {X 0,Y 393.564,Z 278.708,A -85,B 0,C 180,E1 19467.377,E2 19467.377} C_VEL
LIN {X 0,Y 393.565,Z 278.7,A -85,B 0,C 180,E1 19463.349,E2 19463.349} C_VEL
LIN {X 0,Y 393.564,Z 278.699,A -85,B 0,C 180,E1 19459.44,E2 19459.44} C_VEL
LIN {X 0,Y 393.569,Z 278.699,A -85,B 0,C 180,E1 19455.471,E2 19455.471} C_VEL
LIN {X 0,Y 393.56,Z 278.701,A -85,B 0,C 180,E1 19451.43,E2 19451.43} C_VEL
LIN {X 0,Y 393.57,Z 278.705,A -85,B 0,C 180,E1 19447.445,E2 19447.445} C_VEL
LIN {X 0,Y 393.553,Z 278.712,A -85,B 0,C 180,E1 19443.35,E2 19443.35} C_VEL
LIN {X 0,Y 393.561,Z 278.712,A -85,B 0,C 180,E1 19439.418,E2 19439.418} C_VEL
LIN {X 0,Y 393.546,Z 278.711,A -85,B 0,C 180,E1 19435.337,E2 19435.337} C_VEL
LIN {X 0,Y 393.543,Z 278.706,A -85,B 0,C 180,E1 19431.379,E2 19431.379} C_VEL
LIN {X 0,Y 393.537,Z 278.704,A -85,B 0,C 180,E1 19427.317,E2 19427.317} C_VEL
LIN {X 0,Y 393.529,Z 278.704,A -85,B 0,C 180,E1 19423.316,E2 19423.316} C_VEL
LIN {X 0,Y 393.541,Z 278.708,A -85,B 0,C 180,E1 19419.218,E2 19419.218} C_VEL
LIN {X 0,Y 393.544,Z 278.716,A -85,B 0,C 180,E1 19415.216,E2 19415.216} C_VEL
LIN {X 0,Y 393.555,Z 278.696,A -85,B 0,C 180,E1 19411.138,E2 19411.138} C_VEL
LIN {X 0,Y 393.555,Z 278.911,A -85,B 0,C 180,E1 19407.616,E2 19407.616} C_VEL
LIN {X 0,Y 395.034,Z 282.454,A -85,B 0,C 180,E1 19406.685,E2 19406.685} C_VEL
LIN {X 0,Y 396.435,Z 284.782,A -85,B 0,C 180,E1 19406.074,E2 19406.074} C_VEL
LIN {X 0,Y 399.196,Z 289.981,A -85,B 0,C 180,E1 19404.825,E2 19404.825} C_VEL
LIN {X 0,Y 401.824,Z 294.901,A -85,B 0,C 180,E1 19403.686,E2 19403.686} C_VEL
LIN {X 0,Y 407.643,Z 306.259,A -85,B 0,C 180,E1 19401.257,E2 19401.257} C_VEL
LIN {X 0,Y 409.494,Z 309.365,A -85,B 0,C 180,E1 19400.773,E2 19400.773} C_VEL
LIN {X 0,Y 420.187,Z 325.211,A -85,B 0,C 180,E1 19398.766,E2 19398.766} C_VEL
LIN {X 0,Y 431.579,Z 343.598,A -85,B 0,C 180,E1 19396.774,E2 19396.774} C_VEL
LIN {X 0,Y 434.669,Z 349.312,A -85,B 0,C 180,E1 19396.245,E2 19396.245} C_VEL
LIN {X 0,Y 427.116,Z 558.059,A -85,B 0,C 180,E1 19392.32,E2 19392.32} C_VEL
LIN {X 0,Y 425.218,Z 607.206,A -85,B 0,C 180,E1 19391.355,E2 19391.355} C_VEL
LIN {X 0,Y 423.439,Z 629.466,A -85,B 0,C 180,E1 19390.7,E2 19390.7} C_VEL
LIN {X 0,Y 421.284,Z 650.286,A -85,B 0,C 180,E1 19389.851,E2 19389.851} C_VEL
LIN {X 0,Y 418.824,Z 670.41,A -85,B 0,C 180,E1 19388.803,E2 19388.803} C_VEL
LIN {X 0,Y 415.957,Z 690.332,A -85,B 0,C 180,E1 19387.511,E2 19387.511} C_VEL
LIN {X 0,Y 412.84,Z 709.877,A -85,B 0,C 180,E1 19385.965,E2 19385.965} C_VEL
LIN {X 0,Y 409.605,Z 729.005,A -85,B 0,C 180,E1 19384.154,E2 19384.154} C_VEL
LIN {X 0,Y 406.353,Z 747.276,A -85,B 0,C 180,E1 19382.105,E2 19382.105} C_VEL
LIN {X 0,Y 403.165,Z 764.707,A -85,B 0,C 180,E1 19379.773,E2 19379.773} C_VEL
LIN {X 0,Y 400.405,Z 780.077,A -85,B 0,C 180,E1 19377.352,E2 19377.352} C_VEL
LIN {X 0,Y 397.901,Z 794.712,A -85,B 0,C 180,E1 19374.653,E2 19374.653} C_VEL
LIN {X 0,Y 395.939,Z 807.219,A -85,B 0,C 180,E1 19371.946,E2 19371.946} C_VEL
LIN {X 0,Y 394.379,Z 818.26,A -85,B 0,C 180,E1 19369.089,E2 19369.089} C_VEL
LIN {X 0,Y 393.233,Z 828.101,A -85,B 0,C 180,E1 19366.029,E2 19366.029} C_VEL
LIN {X 0,Y 392.54,Z 835.778,A -85,B 0,C 180,E1 19363.102,E2 19363.102} C_VEL
LIN {X 0,Y 392.158,Z 841.76,A -85,B 0,C 180,E1 19360.132,E2 19360.132} C_VEL
LIN {X 0,Y 392.002,Z 846.377,A -85,B 0,C 180,E1 19357.032,E2 19357.032} C_VEL
LIN {X 0,Y 391.954,Z 849.092,A -85,B 0,C 180,E1 19354.242,E2 19354.242} C_VEL
LIN {X 0,Y 391.957,Z 850.503,A -85,B 0,C 180,E1 19351.169,E2 19351.169} C_VEL
LIN {X 0,Y 391.949,Z 850.429,A -85,B 0,C 180,E1 19348.392,E2 19348.392} C_VEL
LIN {X 0,Y 391.959,Z 848.735,A -85,B 0,C 180,E1 19345.318,E2 19345.318} C_VEL
LIN {X 0,Y 392.009,Z 845.686,A -85,B 0,C 180,E1 19342.379,E2 19342.379} C_VEL
LIN {X 0,Y 392.207,Z 840.967,A -85,B 0,C 180,E1 19339.424,E2 19339.424} C_VEL
LIN {X 0,Y 392.653,Z 834.323,A -85,B 0,C 180,E1 19336.302,E2 19336.302} C_VEL
LIN {X 0,Y 393.444,Z 826.214,A -85,B 0,C 180,E1 19333.312,E2 19333.312} C_VEL
LIN {X 0,Y 394.596,Z 816.625,A -85,B 0,C 180,E1 19330.46,E2 19330.46} C_VEL
LIN {X 0,Y 396.347,Z 804.381,A -85,B 0,C 180,E1 19327.413,E2 19327.413} C_VEL
LIN {X 0,Y 398.407,Z 791.716,A -85,B 0,C 180,E1 19324.746,E2 19324.746} C_VEL
LIN {X 0,Y 400.878,Z 777.426,A -85,B 0,C 180,E1 19322.199,E2 19322.199} C_VEL
LIN {X 0,Y 403.7,Z 761.746,A -85,B 0,C 180,E1 19319.812,E2 19319.812} C_VEL
LIN {X 0,Y 406.773,Z 744.766,A -85,B 0,C 180,E1 19317.6,E2 19317.6} C_VEL
LIN {X 0,Y 410.114,Z 726.223,A -85,B 0,C 180,E1 19315.556,E2 19315.556} C_VEL
LIN {X 0,Y 413.25,Z 707.357,A -85,B 0,C 180,E1 19313.819,E2 19313.819} C_VEL
LIN {X 0,Y 416.36,Z 687.537,A -85,B 0,C 180,E1 19312.297,E2 19312.297} C_VEL
LIN {X 0,Y 419.184,Z 667.651,A -85,B 0,C 180,E1 19311.04,E2 19311.04} C_VEL
LIN {X 0,Y 421.681,Z 646.689,A -85,B 0,C 180,E1 19309.984,E2 19309.984} C_VEL
LIN {X 0,Y 423.802,Z 625.032,A -85,B 0,C 180,E1 19309.156,E2 19309.156} C_VEL
LIN {X 0,Y 425.48,Z 602.082,A -85,B 0,C 180,E1 19308.535,E2 19308.535} C_VEL
LIN {X 0,Y 433.082,Z 392.632,A -85,B 0,C 180,E1 19304.569,E2 19304.569} C_VEL
LIN {X 0,Y 434.591,Z 348.79,A -85,B 0,C 180,E1 19303.737,E2 19303.737} C_VEL
LIN {X 0,Y 422.434,Z 328.616,A -85,B 0,C 180,E1 19301.644,E2 19301.644} C_VEL
LIN {X 0,Y 410.912,Z 311.427,A -85,B 0,C 180,E1 19299.516,E2 19299.516} C_VEL
LIN {X 0,Y 407.903,Z 306.874,A -85,B 0,C 180,E1 19298.866,E2 19298.866} C_VEL
LIN {X 0,Y 402.105,Z 295.487,A -85,B 0,C 180,E1 19296.462,E2 19296.462} C_VEL
LIN {X 0,Y 400.123,Z 291.753,A -85,B 0,C 180,E1 19295.608,E2 19295.608} C_VEL
LIN {X 0,Y 397.878,Z 287.482,A -85,B 0,C 180,E1 19294.606,E2 19294.606} C_VEL
LIN {X 0,Y 395.71,Z 283.304,A -85,B 0,C 180,E1 19293.597,E2 19293.597} C_VEL
LIN {X 0,Y 393.839,Z 280.042,A -85,B 0,C 180,E1 19292.735,E2 19292.735} C_VEL
LIN {X 0,Y 393.551,Z 278.868,A -85,B 0,C 180,E1 19292.416,E2 19292.416} C_VEL
LIN {X 0,Y 393.557,Z 278.698,A -85,B 0,C 180,E1 19288.78,E2 19288.78} C_VEL
LIN {X 0,Y 393.545,Z 278.716,A -85,B 0,C 180,E1 19284.784,E2 19284.784} C_VEL
LIN {X 0,Y 393.543,Z 278.708,A -85,B 0,C 180,E1 19280.782,E2 19280.782} C_VEL
LIN {X 0,Y 393.534,Z 278.704,A -85,B 0,C 180,E1 19276.684,E2 19276.684} C_VEL
LIN {X 0,Y 393.533,Z 278.706,A -85,B 0,C 180,E1 19272.77,E2 19272.77} C_VEL
LIN {X 0,Y 393.539,Z 278.71,A -85,B 0,C 180,E1 19268.768,E2 19268.768} C_VEL
LIN {X 0,Y 393.537,Z 278.715,A -85,B 0,C 180,E1 19264.809,E2 19264.809} C_VEL
LIN {X 0,Y 393.55,Z 278.715,A -85,B 0,C 180,E1 19260.728,E2 19260.728} C_VEL
LIN {X 0,Y 393.542,Z 278.711,A -85,B 0,C 180,E1 19256.796,E2 19256.796} C_VEL
LIN {X 0,Y 393.545,Z 278.703,A -85,B 0,C 180,E1 19252.848,E2 19252.848} C_VEL
LIN {X 0,Y 393.541,Z 278.698,A -85,B 0,C 180,E1 19248.866,E2 19248.866} C_VEL
LIN {X 0,Y 393.545,Z 278.697,A -85,B 0,C 180,E1 19244.888,E2 19244.888} C_VEL
LIN {X 0,Y 393.544,Z 278.697,A -85,B 0,C 180,E1 19240.926,E2 19240.926} C_VEL
LIN {X 0,Y 393.544,Z 278.698,A -85,B 0,C 180,E1 19236.967,E2 19236.967} C_VEL
LIN {X 0,Y 393.549,Z 278.703,A -85,B 0,C 180,E1 19232.949,E2 19232.949} C_VEL
LIN {X 0,Y 393.539,Z 278.652,A -85,B 0,C 180,E1 19229.121,E2 19229.121} C_VEL
LIN {X 0,Y 393.547,Z 278.7,A -85,B 0,C 180,E1 19225.135,E2 19225.135} C_VEL
LIN {X 0,Y 393.626,Z 279.113,A -85,B 0,C 180,E1 19224.276,E2 19224.276} C_VEL
LIN {X 0,Y 395.251,Z 282.695,A -85,B 0,C 180,E1 19223.344,E2 19223.344} C_VEL
LIN {X 0,Y 396.252,Z 284.43,A -85,B 0,C 180,E1 19222.877,E2 19222.877} C_VEL
LIN {X 0,Y 398.907,Z 289.767,A -85,B 0,C 180,E1 19221.566,E2 19221.566} C_VEL
LIN {X 0,Y 402.776,Z 297.145,A -85,B 0,C 180,E1 19219.802,E2 19219.802} C_VEL
LIN {X 0,Y 408.976,Z 310.578,A -85,B 0,C 180,E1 19216.968,E2 19216.968} C_VEL
LIN {X 0,Y 415.051,Z 324.305,A -85,B 0,C 180,E1 19214.392,E2 19214.392} C_VEL
LIN {X 0,Y 426.548,Z 343.247,A -85,B 0,C 180,E1 19212.331,E2 19212.331} C_VEL
LIN {X 0,Y 428.313,Z 346.751,A -85,B 0,C 180,E1 19212.018,E2 19212.018} C_VEL
LIN {X 0,Y 431.321,Z 367.666,A -85,B 0,C 180,E1 19211.169,E2 19211.169} C_VEL
LIN {X 0,Y 424.795,Z 594.843,A -85,B 0,C 180,E1 19207.216,E2 19207.216} C_VEL
LIN {X 0,Y 423.409,Z 615.362,A -85,B 0,C 180,E1 19206.633,E2 19206.633} C_VEL
LIN {X 0,Y 421.543,Z 634.603,A -85,B 0,C 180,E1 19205.863,E2 19205.863} C_VEL
LIN {X 0,Y 419.178,Z 653.943,A -85,B 0,C 180,E1 19204.846,E2 19204.846} C_VEL
LIN {X 0,Y 416.427,Z 672.758,A -85,B 0,C 180,E1 19203.594,E2 19203.594} C_VEL
LIN {X 0,Y 413.301,Z 691.116,A -85,B 0,C 180,E1 19202.073,E2 19202.073} C_VEL
LIN {X 0,Y 410.128,Z 707.799,A -85,B 0,C 180,E1 19200.388,E2 19200.388} C_VEL
LIN {X 0,Y 406.912,Z 723.665,A -85,B 0,C 180,E1 19198.469,E2 19198.469} C_VEL
LIN {X 0,Y 406.727,Z 724.539,A -85,B 0,C 180,E1 19198.353,E2 19198.353} C_VEL
LIN {X 0,Y 404.659,Z 730.21,A -85,B 0,C 180,E1 19197.653,E2 19197.653} C_VEL
LIN {X 0,Y 396.3,Z 744.103,A -85,B 0,C 180,E1 19195.941,E2 19195.941} C_VEL
LIN {X 0,Y 394.299,Z 749.009,A -85,B 0,C 180,E1 19195.133,E2 19195.133} C_VEL
LIN {X 0,Y 391.391,Z 761.933,A -85,B 0,C 180,E1 19192.531,E2 19192.531} C_VEL
LIN {X 0,Y 389.012,Z 773.056,A -85,B 0,C 180,E1 19189.828,E2 19189.828} C_VEL
LIN {X 0,Y 387.117,Z 782.732,A -85,B 0,C 180,E1 19186.969,E2 19186.969} C_VEL
LIN {X 0,Y 385.723,Z 790.918,A -85,B 0,C 180,E1 19183.949,E2 19183.949} C_VEL
LIN {X 0,Y 384.835,Z 797.246,A -85,B 0,C 180,E1 19180.933,E2 19180.933} C_VEL
LIN {X 0,Y 384.349,Z 801.936,A -85,B 0,C 180,E1 19177.925,E2 19177.925} C_VEL
LIN {X 0,Y 384.126,Z 805.115,A -85,B 0,C 180,E1 19174.927,E2 19174.927} C_VEL
LIN {X 0,Y 384.048,Z 806.799,A -85,B 0,C 180,E1 19171.94,E2 19171.94} C_VEL
LIN {X 0,Y 384.037,Z 807.002,A -85,B 0,C 180,E1 19168.956,E2 19168.956} C_VEL
LIN {X 0,Y 384.09,Z 805.714,A -85,B 0,C 180,E1 19165.82,E2 19165.82} C_VEL
LIN {X 0,Y 384.269,Z 803.029,A -85,B 0,C 180,E1 19162.826,E2 19162.826} C_VEL
LIN {X 0,Y 384.698,Z 798.503,A -85,B 0,C 180,E1 19159.669,E2 19159.669} C_VEL
LIN {X 0,Y 385.493,Z 792.313,A -85,B 0,C 180,E1 19156.568,E2 19156.568} C_VEL
LIN {X 0,Y 386.785,Z 784.499,A -85,B 0,C 180,E1 19153.548,E2 19153.548} C_VEL
LIN {X 0,Y 388.61,Z 775.014,A -85,B 0,C 180,E1 19150.616,E2 19150.616} C_VEL
LIN {X 0,Y 390.879,Z 764.352,A -85,B 0,C 180,E1 19147.913,E2 19147.913} C_VEL
LIN {X 0,Y 393.582,Z 752.311,A -85,B 0,C 180,E1 19145.379,E2 19145.379} C_VEL
LIN {X 0,Y 396.629,Z 738.788,A -85,B 0,C 180,E1 19143.016,E2 19143.016} C_VEL
LIN {X 0,Y 399.972,Z 723.825,A -85,B 0,C 180,E1 19140.827,E2 19140.827} C_VEL
LIN {X 0,Y 403.483,Z 707.261,A -85,B 0,C 180,E1 19138.808,E2 19138.808} C_VEL
LIN {X 0,Y 406.831,Z 690.372,A -85,B 0,C 180,E1 19137.103,E2 19137.103} C_VEL
LIN {X 0,Y 409.979,Z 672.682,A -85,B 0,C 180,E1 19135.628,E2 19135.628} C_VEL
LIN {X 0,Y 412.829,Z 653.997,A -85,B 0,C 180,E1 19134.376,E2 19134.376} C_VEL
LIN {X 0,Y 415.233,Z 635.17,A -85,B 0,C 180,E1 19133.377,E2 19133.377} C_VEL
LIN {X 0,Y 417.255,Z 615.142,A -85,B 0,C 180,E1 19132.568,E2 19132.568} C_VEL
LIN {X 0,Y 418.689,Z 594.734,A -85,B 0,C 180,E1 19131.986,E2 19131.986} C_VEL
LIN {X 0,Y 425.539,Z 367.853,A -85,B 0,C 180,E1 19127.981,E2 19127.981} C_VEL
LIN {X 0,Y 422.677,Z 349.873,A -85,B 0,C 180,E1 19127.191,E2 19127.191} C_VEL
LIN {X 0,Y 412.517,Z 332.852,A -85,B 0,C 180,E1 19125.335,E2 19125.335} C_VEL
LIN {X 0,Y 406.319,Z 322.811,A -85,B 0,C 180,E1 19124.067,E2 19124.067} C_VEL
LIN {X 0,Y 400.038,Z 308.844,A -85,B 0,C 180,E1 19121.21,E2 19121.21} C_VEL
LIN {X 0,Y 394.835,Z 297.878,A -85,B 0,C 180,E1 19118.718,E2 19118.718} C_VEL
LIN {X 0,Y 389.939,Z 288.512,A -85,B 0,C 180,E1 19116.322,E2 19116.322} C_VEL
LIN {X 0,Y 387.619,Z 284.071,A -85,B 0,C 180,E1 19115.116,E2 19115.116} C_VEL
LIN {X 0,Y 385.889,Z 280.998,A -85,B 0,C 180,E1 19114.212,E2 19114.212} C_VEL
LIN {X 0,Y 385.651,Z 279.888,A -85,B 0,C 180,E1 19113.878,E2 19113.878} C_VEL
LIN {X 0,Y 385.623,Z 279.646,A -85,B 0,C 180,E1 19110.005,E2 19110.005} C_VEL
LIN {X 0,Y 385.612,Z 279.686,A -85,B 0,C 180,E1 19106.155,E2 19106.155} C_VEL
LIN {X 0,Y 385.603,Z 279.685,A -85,B 0,C 180,E1 19102.231,E2 19102.231} C_VEL
LIN {X 0,Y 385.596,Z 279.685,A -85,B 0,C 180,E1 19098.286,E2 19098.286} C_VEL
LIN {X 0,Y 385.591,Z 279.684,A -85,B 0,C 180,E1 19094.261,E2 19094.261} C_VEL
LIN {X 0,Y 385.585,Z 279.683,A -85,B 0,C 180,E1 19090.307,E2 19090.307} C_VEL
LIN {X 0,Y 385.577,Z 279.686,A -85,B 0,C 180,E1 19086.402,E2 19086.402} C_VEL
LIN {X 0,Y 385.573,Z 279.692,A -85,B 0,C 180,E1 19082.378,E2 19082.378} C_VEL
LIN {X 0,Y 385.568,Z 279.699,A -85,B 0,C 180,E1 19078.366,E2 19078.366} C_VEL
LIN {X 0,Y 385.563,Z 279.706,A -85,B 0,C 180,E1 19074.345,E2 19074.345} C_VEL
LIN {X 0,Y 385.557,Z 279.708,A -85,B 0,C 180,E1 19070.296,E2 19070.296} C_VEL
LIN {X 0,Y 385.551,Z 279.708,A -85,B 0,C 180,E1 19066.197,E2 19066.197} C_VEL
LIN {X 0,Y 385.553,Z 279.707,A -85,B 0,C 180,E1 19062.123,E2 19062.123} C_VEL
LIN {X 0,Y 385.557,Z 279.701,A -85,B 0,C 180,E1 19058.073,E2 19058.073} C_VEL
LIN {X 0,Y 385.566,Z 279.696,A -85,B 0,C 180,E1 19054.135,E2 19054.135} C_VEL
LIN {X 0,Y 385.565,Z 279.66,A -85,B 0,C 180,E1 19050.139,E2 19050.139} C_VEL
LIN {X 0,Y 385.684,Z 280.083,A -85,B 0,C 180,E1 19049.145,E2 19049.145} C_VEL
LIN {X 0,Y 387.2,Z 283.584,A -85,B 0,C 180,E1 19048.212,E2 19048.212} C_VEL
LIN {X 0,Y 388.5,Z 285.517,A -85,B 0,C 180,E1 19047.635,E2 19047.635} C_VEL
LIN {X 0,Y 391.501,Z 291.303,A -85,B 0,C 180,E1 19046.169,E2 19046.169} C_VEL
LIN {X 0,Y 394.028,Z 296.021,A -85,B 0,C 180,E1 19045.007,E2 19045.007} C_VEL
LIN {X 0,Y 398.026,Z 303.537,A -85,B 0,C 180,E1 19043.256,E2 19043.256} C_VEL
LIN {X 0,Y 400.512,Z 308.361,A -85,B 0,C 180,E1 19042.27,E2 19042.27} C_VEL
LIN {X 0,Y 412.364,Z 325.544,A -85,B 0,C 180,E1 19039.905,E2 19039.905} C_VEL
LIN {X 0,Y 423.917,Z 343.854,A -85,B 0,C 180,E1 19037.786,E2 19037.786} C_VEL
LIN {X 0,Y 428.787,Z 352.536,A -85,B 0,C 180,E1 19036.925,E2 19036.925} C_VEL
LIN {X 0,Y 420.884,Z 561.107,A -85,B 0,C 180,E1 19032.961,E2 19032.961} C_VEL
LIN {X 0,Y 419.009,Z 607.146,A -85,B 0,C 180,E1 19032.044,E2 19032.044} C_VEL
LIN {X 0,Y 417.149,Z 629.437,A -85,B 0,C 180,E1 19031.381,E2 19031.381} C_VEL
LIN {X 0,Y 414.852,Z 650.614,A -85,B 0,C 180,E1 19030.505,E2 19030.505} C_VEL
LIN {X 0,Y 412.069,Z 672.016,A -85,B 0,C 180,E1 19029.361,E2 19029.361} C_VEL
LIN {X 0,Y 409.038,Z 692.145,A -85,B 0,C 180,E1 19028.023,E2 19028.023} C_VEL
LIN {X 0,Y 405.739,Z 711.575,A -85,B 0,C 180,E1 19026.433,E2 19026.433} C_VEL
LIN {X 0,Y 402.363,Z 730.342,A -85,B 0,C 180,E1 19024.597,E2 19024.597} C_VEL
LIN {X 0,Y 399.081,Z 747.747,A -85,B 0,C 180,E1 19022.592,E2 19022.592} C_VEL
LIN {X 0,Y 395.901,Z 764.277,A -85,B 0,C 180,E1 19020.337,E2 19020.337} C_VEL
LIN {X 0,Y 393.003,Z 779.436,A -85,B 0,C 180,E1 19017.912,E2 19017.912} C_VEL
LIN {X 0,Y 390.461,Z 793.357,A -85,B 0,C 180,E1 19015.317,E2 19015.317} C_VEL
LIN {X 0,Y 388.222,Z 806.651,A -85,B 0,C 180,E1 19012.393,E2 19012.393} C_VEL
LIN {X 0,Y 386.564,Z 817.637,A -85,B 0,C 180,E1 19009.491,E2 19009.491} C_VEL
LIN {X 0,Y 385.349,Z 827.324,A -85,B 0,C 180,E1 19006.428,E2 19006.428} C_VEL
LIN {X 0,Y 384.587,Z 835.218,A -85,B 0,C 180,E1 19003.378,E2 19003.378} C_VEL
LIN {X 0,Y 384.181,Z 841.255,A -85,B 0,C 180,E1 19000.338,E2 19000.338} C_VEL
LIN {X 0,Y 384.012,Z 845.893,A -85,B 0,C 180,E1 18997.179,E2 18997.179} C_VEL
LIN {X 0,Y 383.964,Z 848.63,A -85,B 0,C 180,E1 18994.331,E2 18994.331} C_VEL
LIN {X 0,Y 383.969,Z 850.053,A -85,B 0,C 180,E1 18991.194,E2 18991.194} C_VEL
LIN {X 0,Y 383.961,Z 849.979,A -85,B 0,C 180,E1 18988.359,E2 18988.359} C_VEL
LIN {X 0,Y 383.967,Z 848.392,A -85,B 0,C 180,E1 18985.37,E2 18985.37} C_VEL
LIN {X 0,Y 384.015,Z 845.382,A -85,B 0,C 180,E1 18982.369,E2 18982.369} C_VEL
LIN {X 0,Y 384.214,Z 840.708,A -85,B 0,C 180,E1 18979.353,E2 18979.353} C_VEL
LIN {X 0,Y 384.646,Z 834.486,A -85,B 0,C 180,E1 18976.318,E2 18976.318} C_VEL
LIN {X 0,Y 385.452,Z 826.464,A -85,B 0,C 180,E1 18973.266,E2 18973.266} C_VEL
LIN {X 0,Y 386.719,Z 816.55,A -85,B 0,C 180,E1 18970.203,E2 18970.203} C_VEL
LIN {X 0,Y 388.432,Z 805.266,A -85,B 0,C 180,E1 18967.288,E2 18967.288} C_VEL
LIN {X 0,Y 390.737,Z 791.876,A -85,B 0,C 180,E1 18964.377,E2 18964.377} C_VEL
LIN {X 0,Y 393.334,Z 777.665,A -85,B 0,C 180,E1 18961.784,E2 18961.784} C_VEL
LIN {X 0,Y 396.31,Z 762.096,A -85,B 0,C 180,E1 18959.351,E2 18959.351} C_VEL
LIN {X 0,Y 399.534,Z 745.31,A -85,B 0,C 180,E1 18957.109,E2 18957.109} C_VEL
LIN {X 0,Y 402.88,Z 727.612,A -85,B 0,C 180,E1 18955.114,E2 18955.114} C_VEL
LIN {X 0,Y 406.16,Z 709.05,A -85,B 0,C 180,E1 18953.348,E2 18953.348} C_VEL
LIN {X 0,Y 409.563,Z 688.609,A -85,B 0,C 180,E1 18951.731,E2 18951.731} C_VEL
LIN {X 0,Y 412.623,Z 668.193,A -85,B 0,C 180,E1 18950.411,E2 18950.411} C_VEL
LIN {X 0,Y 415.266,Z 646.978,A -85,B 0,C 180,E1 18949.327,E2 18949.327} C_VEL
LIN {X 0,Y 417.523,Z 625.086,A -85,B 0,C 180,E1 18948.477,E2 18948.477} C_VEL
LIN {X 0,Y 419.255,Z 602.502,A -85,B 0,C 180,E1 18947.855,E2 18947.855} C_VEL
LIN {X 0,Y 427.131,Z 395.583,A -85,B 0,C 180,E1 18943.893,E2 18943.893} C_VEL
LIN {X 0,Y 428.631,Z 351.994,A -85,B 0,C 180,E1 18943.047,E2 18943.047} C_VEL
LIN {X 0,Y 417.089,Z 332.854,A -85,B 0,C 180,E1 18940.991,E2 18940.991} C_VEL
LIN {X 0,Y 405.666,Z 315.671,A -85,B 0,C 180,E1 18938.804,E2 18938.804} C_VEL
LIN {X 0,Y 399.979,Z 307.34,A -85,B 0,C 180,E1 18937.585,E2 18937.585} C_VEL
LIN {X 0,Y 394.815,Z 297.507,A -85,B 0,C 180,E1 18935.37,E2 18935.37} C_VEL
LIN {X 0,Y 392.396,Z 292.963,A -85,B 0,C 180,E1 18934.272,E2 18934.272} C_VEL
LIN {X 0,Y 390.244,Z 288.869,A -85,B 0,C 180,E1 18933.25,E2 18933.25} C_VEL
LIN {X 0,Y 387.85,Z 284.363,A -85,B 0,C 180,E1 18932.077,E2 18932.077} C_VEL
LIN {X 0,Y 385.994,Z 281.334,A -85,B 0,C 180,E1 18931.202,E2 18931.202} C_VEL
LIN {X 0,Y 385.639,Z 279.852,A -85,B 0,C 180,E1 18930.774,E2 18930.774} C_VEL
LIN {X 0,Y 385.609,Z 279.688,A -85,B 0,C 180,E1 18926.818,E2 18926.818} C_VEL
LIN {X 0,Y 385.608,Z 279.686,A -85,B 0,C 180,E1 18922.727,E2 18922.727} C_VEL
LIN {X 0,Y 385.596,Z 279.687,A -85,B 0,C 180,E1 18918.755,E2 18918.755} C_VEL
LIN {X 0,Y 385.605,Z 279.686,A -85,B 0,C 180,E1 18914.721,E2 18914.721} C_VEL
LIN {X 0,Y 385.59,Z 279.689,A -85,B 0,C 180,E1 18910.609,E2 18910.609} C_VEL
LIN {X 0,Y 385.603,Z 279.686,A -85,B 0,C 180,E1 18906.551,E2 18906.551} C_VEL
LIN {X 0,Y 385.601,Z 279.684,A -85,B 0,C 180,E1 18902.526,E2 18902.526} C_VEL
LIN {X 0,Y 385.611,Z 279.682,A -85,B 0,C 180,E1 18898.514,E2 18898.514} C_VEL
LIN {X 0,Y 385.614,Z 279.681,A -85,B 0,C 180,E1 18894.494,E2 18894.494} C_VEL
LIN {X 0,Y 385.616,Z 279.684,A -85,B 0,C 180,E1 18890.598,E2 18890.598} C_VEL
LIN {X 0,Y 385.626,Z 279.687,A -85,B 0,C 180,E1 18886.478,E2 18886.478} C_VEL
LIN {X 0,Y 385.623,Z 279.69,A -85,B 0,C 180,E1 18882.496,E2 18882.496} C_VEL
LIN {X 0,Y 385.632,Z 279.687,A -85,B 0,C 180,E1 18878.397,E2 18878.397} C_VEL
LIN {X 0,Y 385.623,Z 279.685,A -85,B 0,C 180,E1 18874.341,E2 18874.341} C_VEL
LIN {X 0,Y 385.626,Z 279.653,A -85,B 0,C 180,E1 18870.315,E2 18870.315} C_VEL
LIN {X 0,Y 385.629,Z 279.735,A -85,B 0,C 180,E1 18866.299,E2 18866.299} C_VEL
LIN {X 0,Y 385.704,Z 280.234,A -85,B 0,C 180,E1 18865.859,E2 18865.859} C_VEL
LIN {X 0,Y 387.382,Z 283.785,A -85,B 0,C 180,E1 18864.86,E2 18864.86} C_VEL
LIN {X 0,Y 388.315,Z 285.273,A -85,B 0,C 180,E1 18864.414,E2 18864.414} C_VEL
LIN {X 0,Y 391.26,Z 291.166,A -85,B 0,C 180,E1 18862.872,E2 18862.872} C_VEL
LIN {X 0,Y 393.642,Z 295.805,A -85,B 0,C 180,E1 18861.701,E2 18861.701} C_VEL
LIN {X 0,Y 399.057,Z 306.585,A -85,B 0,C 180,E1 18859.16,E2 18859.16} C_VEL
LIN {X 0,Y 405.959,Z 321.987,A -85,B 0,C 180,E1 18855.985,E2 18855.985} C_VEL
LIN {X 0,Y 407.473,Z 324.894,A -85,B 0,C 180,E1 18855.528,E2 18855.528} C_VEL
LIN {X 0,Y 418.592,Z 342.875,A -85,B 0,C 180,E1 18853.436,E2 18853.436} C_VEL
LIN {X 0,Y 422.946,Z 350.72,A -85,B 0,C 180,E1 18852.649,E2 18852.649} C_VEL
LIN {X 0,Y 425.51,Z 369.317,A -85,B 0,C 180,E1 18851.886,E2 18851.886} C_VEL
LIN {X 0,Y 418.644,Z 595.025,A -85,B 0,C 180,E1 18847.912,E2 18847.912} C_VEL
LIN {X 0,Y 417.188,Z 615.637,A -85,B 0,C 180,E1 18847.321,E2 18847.321} C_VEL
LIN {X 0,Y 415.231,Z 634.969,A -85,B 0,C 180,E1 18846.538,E2 18846.538} C_VEL
LIN {X 0,Y 412.792,Z 654.057,A -85,B 0,C 180,E1 18845.525,E2 18845.525} C_VEL
LIN {X 0,Y 409.979,Z 672.547,A -85,B 0,C 180,E1 18844.288,E2 18844.288} C_VEL
LIN {X 0,Y 406.798,Z 690.434,A -85,B 0,C 180,E1 18842.797,E2 18842.797} C_VEL
LIN {X 0,Y 403.431,Z 707.423,A -85,B 0,C 180,E1 18841.078,E2 18841.078} C_VEL
LIN {X 0,Y 400.01,Z 723.568,A -85,B 0,C 180,E1 18839.113,E2 18839.113} C_VEL
LIN {X 0,Y 396.738,Z 738.258,A -85,B 0,C 180,E1 18836.976,E2 18836.976} C_VEL
LIN {X 0,Y 394.299,Z 749.009,A -85,B 0,C 180,E1 18835.133,E2 18835.133} C_VEL
LIN {X 0,Y 392.315,Z 753.864,A -85,B 0,C 180,E1 18834.293,E2 18834.293} C_VEL
LIN {X 0,Y 384.107,Z 765.637,A -85,B 0,C 180,E1 18832.202,E2 18832.202} C_VEL
LIN {X 0,Y 382.257,Z 769.688,A -85,B 0,C 180,E1 18831.261,E2 18831.261} C_VEL
LIN {X 0,Y 380.044,Z 779.848,A -85,B 0,C 180,E1 18828.403,E2 18828.403} C_VEL
LIN {X 0,Y 378.404,Z 788.33,A -85,B 0,C 180,E1 18825.478,E2 18825.478} C_VEL
LIN {X 0,Y 377.243,Z 795.431,A -85,B 0,C 180,E1 18822.397,E2 18822.397} C_VEL
LIN {X 0,Y 376.544,Z 800.968,A -85,B 0,C 180,E1 18819.167,E2 18819.167} C_VEL
LIN {X 0,Y 376.208,Z 804.611,A -85,B 0,C 180,E1 18816.102,E2 18816.102} C_VEL
LIN {X 0,Y 376.073,Z 806.867,A -85,B 0,C 180,E1 18812.895,E2 18812.895} C_VEL
LIN {X 0,Y 376.052,Z 807.578,A -85,B 0,C 180,E1 18809.848,E2 18809.848} C_VEL
LIN {X 0,Y 376.075,Z 806.782,A -85,B 0,C 180,E1 18806.799,E2 18806.799} C_VEL
LIN {X 0,Y 376.218,Z 804.518,A -85,B 0,C 180,E1 18803.704,E2 18803.704} C_VEL
LIN {X 0,Y 376.578,Z 800.638,A -85,B 0,C 180,E1 18800.525,E2 18800.525} C_VEL
LIN {X 0,Y 377.266,Z 795.308,A -85,B 0,C 180,E1 18797.449,E2 18797.449} C_VEL
LIN {X 0,Y 378.436,Z 788.181,A -85,B 0,C 180,E1 18794.366,E2 18794.366} C_VEL
LIN {X 0,Y 380.09,Z 779.654,A -85,B 0,C 180,E1 18791.44,E2 18791.44} C_VEL
LIN {X 0,Y 382.368,Z 769.221,A -85,B 0,C 180,E1 18788.526,E2 18788.526} C_VEL
LIN {X 0,Y 385.161,Z 757.285,A -85,B 0,C 180,E1 18785.786,E2 18785.786} C_VEL
LIN {X 0,Y 388.245,Z 744.472,A -85,B 0,C 180,E1 18783.335,E2 18783.335} C_VEL
LIN {X 0,Y 391.842,Z 729.308,A -85,B 0,C 180,E1 18780.928,E2 18780.928} C_VEL
LIN {X 0,Y 395.367,Z 713.783,A -85,B 0,C 180,E1 18778.891,E2 18778.891} C_VEL
LIN {X 0,Y 398.924,Z 696.977,A -85,B 0,C 180,E1 18777.052,E2 18777.052} C_VEL
LIN {X 0,Y 402.45,Z 678.736,A -85,B 0,C 180,E1 18775.412,E2 18775.412} C_VEL
LIN {X 0,Y 405.561,Z 660.456,A -85,B 0,C 180,E1 18774.074,E2 18774.074} C_VEL
LIN {X 0,Y 408.28,Z 641.297,A -85,B 0,C 180,E1 18772.956,E2 18772.956} C_VEL
LIN {X 0,Y 410.531,Z 621.409,A -85,B 0,C 180,E1 18772.077,E2 18772.077} C_VEL
LIN {X 0,Y 412.204,Z 601.034,A -85,B 0,C 180,E1 18771.426,E2 18771.426} C_VEL
LIN {X 0,Y 413.311,Z 576.324,A -85,B 0,C 180,E1 18770.915,E2 18770.915} C_VEL
LIN {X 0,Y 419.795,Z 369.241,A -85,B 0,C 180,E1 18767.237,E2 18767.237} C_VEL
LIN {X 0,Y 417.446,Z 354.07,A -85,B 0,C 180,E1 18766.558,E2 18766.558} C_VEL
LIN {X 0,Y 406.213,Z 335.182,A -85,B 0,C 180,E1 18764.425,E2 18764.425} C_VEL
LIN {X 0,Y 398.28,Z 322.781,A -85,B 0,C 180,E1 18762.772,E2 18762.772} C_VEL
LIN {X 0,Y 392.308,Z 309.815,A -85,B 0,C 180,E1 18759.961,E2 18759.961} C_VEL
LIN {X 0,Y 387.133,Z 299.071,A -85,B 0,C 180,E1 18757.369,E2 18757.369} C_VEL
LIN {X 0,Y 384.104,Z 293.492,A -85,B 0,C 180,E1 18755.853,E2 18755.853} C_VEL
LIN {X 0,Y 382.45,Z 290.062,A -85,B 0,C 180,E1 18754.928,E2 18754.928} C_VEL
LIN {X 0,Y 380.485,Z 286.392,A -85,B 0,C 180,E1 18753.856,E2 18753.856} C_VEL
LIN {X 0,Y 377.934,Z 281.916,A -85,B 0,C 180,E1 18752.444,E2 18752.444} C_VEL
LIN {X 0,Y 377.713,Z 280.895,A -85,B 0,C 180,E1 18752.107,E2 18752.107} C_VEL
LIN {X 0,Y 377.669,Z 280.678,A -85,B 0,C 180,E1 18748.46,E2 18748.46} C_VEL
LIN {X 0,Y 377.666,Z 280.694,A -85,B 0,C 180,E1 18744.394,E2 18744.394} C_VEL
LIN {X 0,Y 377.66,Z 280.693,A -85,B 0,C 180,E1 18740.415,E2 18740.415} C_VEL
LIN {X 0,Y 377.655,Z 280.694,A -85,B 0,C 180,E1 18736.299,E2 18736.299} C_VEL
LIN {X 0,Y 377.652,Z 280.693,A -85,B 0,C 180,E1 18732.228,E2 18732.228} C_VEL
LIN {X 0,Y 377.648,Z 280.693,A -85,B 0,C 180,E1 18728.22,E2 18728.22} C_VEL
LIN {X 0,Y 377.64,Z 280.692,A -85,B 0,C 180,E1 18724.252,E2 18724.252} C_VEL
LIN {X 0,Y 377.634,Z 280.684,A -85,B 0,C 180,E1 18720.304,E2 18720.304} C_VEL
LIN {X 0,Y 377.628,Z 280.681,A -85,B 0,C 180,E1 18716.205,E2 18716.205} C_VEL
LIN {X 0,Y 377.62,Z 280.678,A -85,B 0,C 180,E1 18712.24,E2 18712.24} C_VEL
LIN {X 0,Y 377.614,Z 280.676,A -85,B 0,C 180,E1 18708.236,E2 18708.236} C_VEL
LIN {X 0,Y 377.608,Z 280.677,A -85,B 0,C 180,E1 18704.173,E2 18704.173} C_VEL
LIN {X 0,Y 377.615,Z 280.679,A -85,B 0,C 180,E1 18700.189,E2 18700.189} C_VEL
LIN {X 0,Y 377.623,Z 280.684,A -85,B 0,C 180,E1 18696.102,E2 18696.102} C_VEL
LIN {X 0,Y 377.63,Z 280.695,A -85,B 0,C 180,E1 18692.054,E2 18692.054} C_VEL
LIN {X 0,Y 377.736,Z 281.132,A -85,B 0,C 180,E1 18690.908,E2 18690.908} C_VEL
LIN {X 0,Y 379.217,Z 284.525,A -85,B 0,C 180,E1 18689.937,E2 18689.937} C_VEL
LIN {X 0,Y 380.533,Z 286.182,A -85,B 0,C 180,E1 18689.354,E2 18689.354} C_VEL
LIN {X 0,Y 382.478,Z 290.03,A -85,B 0,C 180,E1 18688.302,E2 18688.302} C_VEL
LIN {X 0,Y 386.367,Z 297.316,A -85,B 0,C 180,E1 18686.372,E2 18686.372} C_VEL
LIN {X 0,Y 390.812,Z 305.667,A -85,B 0,C 180,E1 18684.316,E2 18684.316} C_VEL
LIN {X 0,Y 392.765,Z 309.087,A -85,B 0,C 180,E1 18683.597,E2 18683.597} C_VEL
LIN {X 0,Y 404.905,Z 326.442,A -85,B 0,C 180,E1 18681.041,E2 18681.041} C_VEL
LIN {X 0,Y 416.815,Z 345.112,A -85,B 0,C 180,E1 18678.748,E2 18678.748} C_VEL
LIN {X 0,Y 422.96,Z 355.967,A -85,B 0,C 180,E1 18677.62,E2 18677.62} C_VEL
LIN {X 0,Y 414.684,Z 564.76,A -85,B 0,C 180,E1 18673.611,E2 18673.611} C_VEL
LIN {X 0,Y 412.85,Z 607.273,A -85,B 0,C 180,E1 18672.748,E2 18672.748} C_VEL
LIN {X 0,Y 410.907,Z 629.618,A -85,B 0,C 180,E1 18672.077,E2 18672.077} C_VEL
LIN {X 0,Y 408.567,Z 650.221,A -85,B 0,C 180,E1 18671.216,E2 18671.216} C_VEL
LIN {X 0,Y 405.801,Z 670.809,A -85,B 0,C 180,E1 18670.113,E2 18670.113} C_VEL
LIN {X 0,Y 402.737,Z 690.252,A -85,B 0,C 180,E1 18668.818,E2 18668.818} C_VEL
LIN {X 0,Y 399.262,Z 709.921,A -85,B 0,C 180,E1 18667.217,E2 18667.217} C_VEL
LIN {X 0,Y 395.528,Z 729.786,A -85,B 0,C 180,E1 18665.263,E2 18665.263} C_VEL
LIN {X 0,Y 392.053,Z 747.236,A -85,B 0,C 180,E1 18663.228,E2 18663.228} C_VEL
LIN {X 0,Y 388.621,Z 764.157,A -85,B 0,C 180,E1 18660.882,E2 18660.882} C_VEL
LIN {X 0,Y 385.468,Z 779.703,A -85,B 0,C 180,E1 18658.338,E2 18658.338} C_VEL
LIN {X 0,Y 382.651,Z 794.235,A -85,B 0,C 180,E1 18655.539,E2 18655.539} C_VEL
LIN {X 0,Y 380.425,Z 806.746,A -85,B 0,C 180,E1 18652.703,E2 18652.703} C_VEL
LIN {X 0,Y 378.689,Z 817.615,A -85,B 0,C 180,E1 18649.752,E2 18649.752} C_VEL
LIN {X 0,Y 377.408,Z 827.205,A -85,B 0,C 180,E1 18646.625,E2 18646.625} C_VEL
LIN {X 0,Y 376.609,Z 835.007,A -85,B 0,C 180,E1 18643.511,E2 18643.511} C_VEL
LIN {X 0,Y 376.189,Z 840.998,A -85,B 0,C 180,E1 18640.412,E2 18640.412} C_VEL
LIN {X 0,Y 376.018,Z 845.586,A -85,B 0,C 180,E1 18637.179,E2 18637.179} C_VEL
LIN {X 0,Y 375.971,Z 848.41,A -85,B 0,C 180,E1 18634.117,E2 18634.117} C_VEL
LIN {X 0,Y 375.982,Z 849.629,A -85,B 0,C 180,E1 18631.067,E2 18631.067} C_VEL
LIN {X 0,Y 375.973,Z 849.505,A -85,B 0,C 180,E1 18628.171,E2 18628.171} C_VEL
LIN {X 0,Y 375.98,Z 847.804,A -85,B 0,C 180,E1 18625.118,E2 18625.118} C_VEL
LIN {X 0,Y 376.034,Z 844.704,A -85,B 0,C 180,E1 18622.053,E2 18622.053} C_VEL
LIN {X 0,Y 376.249,Z 839.916,A -85,B 0,C 180,E1 18618.97,E2 18618.97} C_VEL
LIN {X 0,Y 376.773,Z 833.192,A -85,B 0,C 180,E1 18615.712,E2 18615.712} C_VEL
LIN {X 0,Y 377.688,Z 825.052,A -85,B 0,C 180,E1 18612.594,E2 18612.594} C_VEL
LIN {X 0,Y 379.104,Z 814.9,A -85,B 0,C 180,E1 18609.466,E2 18609.466} C_VEL
LIN {X 0,Y 380.996,Z 803.349,A -85,B 0,C 180,E1 18606.491,E2 18606.491} C_VEL
LIN {X 0,Y 383.378,Z 790.47,A -85,B 0,C 180,E1 18603.682,E2 18603.682} C_VEL
LIN {X 0,Y 386.18,Z 776.167,A -85,B 0,C 180,E1 18601.043,E2 18601.043} C_VEL
LIN {X 0,Y 389.345,Z 760.458,A -85,B 0,C 180,E1 18598.581,E2 18598.581} C_VEL
LIN {X 0,Y 392.948,Z 742.732,A -85,B 0,C 180,E1 18596.223,E2 18596.223} C_VEL
LIN {X 0,Y 396.516,Z 724.71,A -85,B 0,C 180,E1 18594.197,E2 18594.197} C_VEL
LIN {X 0,Y 400.085,Z 705.457,A -85,B 0,C 180,E1 18592.393,E2 18592.393} C_VEL
LIN {X 0,Y 403.44,Z 685.796,A -85,B 0,C 180,E1 18590.87,E2 18590.87} C_VEL
LIN {X 0,Y 406.549,Z 665.361,A -85,B 0,C 180,E1 18589.572,E2 18589.572} C_VEL
LIN {X 0,Y 409.277,Z 644.449,A -85,B 0,C 180,E1 18588.516,E2 18588.516} C_VEL
LIN {X 0,Y 411.52,Z 623.045,A -85,B 0,C 180,E1 18587.708,E2 18587.708} C_VEL
LIN {X 0,Y 413.243,Z 600.041,A -85,B 0,C 180,E1 18587.093,E2 18587.093} C_VEL
LIN {X 0,Y 421.694,Z 387.19,A -85,B 0,C 180,E1 18582.981,E2 18582.981} C_VEL
LIN {X 0,Y 422.81,Z 355.332,A -85,B 0,C 180,E1 18582.351,E2 18582.351} C_VEL
LIN {X 0,Y 411.429,Z 336.512,A -85,B 0,C 180,E1 18580.25,E2 18580.25} C_VEL
LIN {X 0,Y 399.839,Z 319.053,A -85,B 0,C 180,E1 18577.941,E2 18577.941} C_VEL
LIN {X 0,Y 392.131,Z 308.15,A -85,B 0,C 180,E1 18576.267,E2 18576.267} C_VEL
LIN {X 0,Y 387.058,Z 298.613,A -85,B 0,C 180,E1 18573.984,E2 18573.984} C_VEL
LIN {X 0,Y 384.795,Z 294.375,A -85,B 0,C 180,E1 18572.892,E2 18572.892} C_VEL
LIN {X 0,Y 382.768,Z 290.384,A -85,B 0,C 180,E1 18571.847,E2 18571.847} C_VEL
LIN {X 0,Y 380.709,Z 286.729,A -85,B 0,C 180,E1 18570.805,E2 18570.805} C_VEL
LIN {X 0,Y 379.83,Z 285.235,A -85,B 0,C 180,E1 18570.359,E2 18570.359} C_VEL
LIN {X 0,Y 378.06,Z 282.403,A -85,B 0,C 180,E1 18569.466,E2 18569.466} C_VEL
LIN {X 0,Y 377.701,Z 280.874,A -85,B 0,C 180,E1 18568.976,E2 18568.976} C_VEL
LIN {X 0,Y 377.658,Z 280.692,A -85,B 0,C 180,E1 18565.062,E2 18565.062} C_VEL
LIN {X 0,Y 377.648,Z 280.693,A -85,B 0,C 180,E1 18561.104,E2 18561.104} C_VEL
LIN {X 0,Y 377.64,Z 280.689,A -85,B 0,C 180,E1 18557.091,E2 18557.091} C_VEL
LIN {X 0,Y 377.63,Z 280.693,A -85,B 0,C 180,E1 18553.162,E2 18553.162} C_VEL
LIN {X 0,Y 377.634,Z 280.696,A -85,B 0,C 180,E1 18549.141,E2 18549.141} C_VEL
LIN {X 0,Y 377.629,Z 280.696,A -85,B 0,C 180,E1 18545.317,E2 18545.317} C_VEL
LIN {X 0,Y 377.63,Z 280.692,A -85,B 0,C 180,E1 18541.365,E2 18541.365} C_VEL
LIN {X 0,Y 377.633,Z 280.682,A -85,B 0,C 180,E1 18537.42,E2 18537.42} C_VEL
LIN {X 0,Y 377.636,Z 280.675,A -85,B 0,C 180,E1 18533.462,E2 18533.462} C_VEL
LIN {X 0,Y 377.64,Z 280.672,A -85,B 0,C 180,E1 18529.473,E2 18529.473} C_VEL
LIN {X 0,Y 377.644,Z 280.673,A -85,B 0,C 180,E1 18525.432,E2 18525.432} C_VEL
LIN {X 0,Y 377.652,Z 280.674,A -85,B 0,C 180,E1 18521.406,E2 18521.406} C_VEL
LIN {X 0,Y 377.656,Z 280.674,A -85,B 0,C 180,E1 18517.425,E2 18517.425} C_VEL
LIN {X 0,Y 377.662,Z 280.676,A -85,B 0,C 180,E1 18513.421,E2 18513.421} C_VEL
LIN {X 0,Y 377.658,Z 280.627,A -85,B 0,C 180,E1 18509.364,E2 18509.364} C_VEL
LIN {X 0,Y 377.71,Z 280.926,A -85,B 0,C 180,E1 18507.729,E2 18507.729} C_VEL
LIN {X 0,Y 379.064,Z 284.258,A -85,B 0,C 180,E1 18506.726,E2 18506.726} C_VEL
LIN {X 0,Y 380.338,Z 285.943,A -85,B 0,C 180,E1 18506.129,E2 18506.129} C_VEL
LIN {X 0,Y 382.218,Z 289.776,A -85,B 0,C 180,E1 18505.048,E2 18505.048} C_VEL
LIN {X 0,Y 385.7,Z 296.448,A -85,B 0,C 180,E1 18503.214,E2 18503.214} C_VEL
LIN {X 0,Y 389.943,Z 304.891,A -85,B 0,C 180,E1 18501.082,E2 18501.082} C_VEL
LIN {X 0,Y 395.626,Z 316.941,A -85,B 0,C 180,E1 18498.342,E2 18498.342} C_VEL
LIN {X 0,Y 398.836,Z 323.832,A -85,B 0,C 180,E1 18496.959,E2 18496.959} C_VEL
LIN {X 0,Y 410.48,Z 342.218,A -85,B 0,C 180,E1 18494.637,E2 18494.637} C_VEL
LIN {X 0,Y 417.629,Z 354.686,A -85,B 0,C 180,E1 18493.296,E2 18493.296} C_VEL
LIN {X 0,Y 419.772,Z 370.737,A -85,B 0,C 180,E1 18492.627,E2 18492.627} C_VEL
LIN {X 0,Y 412.556,Z 595.184,A -85,B 0,C 180,E1 18488.629,E2 18488.629} C_VEL
LIN {X 0,Y 411.034,Z 615.816,A -85,B 0,C 180,E1 18488.032,E2 18488.032} C_VEL
LIN {X 0,Y 408.976,Z 635.321,A -85,B 0,C 180,E1 18487.234,E2 18487.234} C_VEL
LIN {X 0,Y 406.381,Z 654.714,A -85,B 0,C 180,E1 18486.191,E2 18486.191} C_VEL
LIN {X 0,Y 403.41,Z 673.307,A -85,B 0,C 180,E1 18484.926,E2 18484.926} C_VEL
LIN {X 0,Y 399.985,Z 691.756,A -85,B 0,C 180,E1 18483.362,E2 18483.362} C_VEL
LIN {X 0,Y 396.499,Z 708.446,A -85,B 0,C 180,E1 18481.635,E2 18481.635} C_VEL
LIN {X 0,Y 392.949,Z 724.361,A -85,B 0,C 180,E1 18479.657,E2 18479.657} C_VEL
LIN {X 0,Y 389.558,Z 738.818,A -85,B 0,C 180,E1 18477.515,E2 18477.515} C_VEL
LIN {X 0,Y 386.342,Z 752.393,A -85,B 0,C 180,E1 18475.114,E2 18475.114} C_VEL
LIN {X 0,Y 383.314,Z 765.144,A -85,B 0,C 180,E1 18472.385,E2 18472.385} C_VEL
LIN {X 0,Y 382.257,Z 769.688,A -85,B 0,C 180,E1 18471.261,E2 18471.261} C_VEL
LIN {X 0,Y 380.461,Z 773.655,A -85,B 0,C 180,E1 18470.292,E2 18470.292} C_VEL
LIN {X 0,Y 372.728,Z 783.089,A -85,B 0,C 180,E1 18467.848,E2 18467.848} C_VEL
LIN {X 0,Y 371.111,Z 786.231,A -85,B 0,C 180,E1 18466.788,E2 18466.788} C_VEL
LIN {X 0,Y 369.668,Z 793.911,A -85,B 0,C 180,E1 18463.61,E2 18463.61} C_VEL
LIN {X 0,Y 368.77,Z 799.999,A -85,B 0,C 180,E1 18460.308,E2 18460.308} C_VEL
LIN {X 0,Y 368.319,Z 804.172,A -85,B 0,C 180,E1 18457.173,E2 18457.173} C_VEL
LIN {X 0,Y 368.121,Z 806.761,A -85,B 0,C 180,E1 18454.049,E2 18454.049} C_VEL
LIN {X 0,Y 368.067,Z 807.906,A -85,B 0,C 180,E1 18450.934,E2 18450.934} C_VEL
LIN {X 0,Y 368.074,Z 807.674,A -85,B 0,C 180,E1 18447.821,E2 18447.821} C_VEL
LIN {X 0,Y 368.173,Z 805.982,A -85,B 0,C 180,E1 18444.702,E2 18444.702} C_VEL
LIN {X 0,Y 368.451,Z 802.781,A -85,B 0,C 180,E1 18441.574,E2 18441.574} C_VEL
LIN {X 0,Y 369.071,Z 797.785,A -85,B 0,C 180,E1 18438.277,E2 18438.277} C_VEL
LIN {X 0,Y 370.134,Z 791.344,A -85,B 0,C 180,E1 18435.13,E2 18435.13} C_VEL
LIN {X 0,Y 371.792,Z 783.082,A -85,B 0,C 180,E1 18431.985,E2 18431.985} C_VEL
LIN {X 0,Y 374.142,Z 772.726,A -85,B 0,C 180,E1 18428.853,E2 18428.853} C_VEL
LIN {X 0,Y 376.899,Z 761.349,A -85,B 0,C 180,E1 18426.054,E2 18426.054} C_VEL
LIN {X 0,Y 380.154,Z 748.387,A -85,B 0,C 180,E1 18423.412,E2 18423.412} C_VEL
LIN {X 0,Y 383.719,Z 734.22,A -85,B 0,C 180,E1 18421.011,E2 18421.011} C_VEL
LIN {X 0,Y 387.312,Z 719.486,A -85,B 0,C 180,E1 18418.916,E2 18418.916} C_VEL
LIN {X 0,Y 391.182,Z 702.645,A -85,B 0,C 180,E1 18416.928,E2 18416.928} C_VEL
LIN {X 0,Y 394.923,Z 684.604,A -85,B 0,C 180,E1 18415.187,E2 18415.187} C_VEL
LIN {X 0,Y 398.087,Z 667.384,A -85,B 0,C 180,E1 18413.827,E2 18413.827} C_VEL
LIN {X 0,Y 401.147,Z 648.123,A -85,B 0,C 180,E1 18412.599,E2 18412.599} C_VEL
LIN {X 0,Y 403.681,Z 628.534,A -85,B 0,C 180,E1 18411.624,E2 18411.624} C_VEL
LIN {X 0,Y 405.732,Z 607.477,A -85,B 0,C 180,E1 18410.859,E2 18410.859} C_VEL
LIN {X 0,Y 406.98,Z 586.509,A -85,B 0,C 180,E1 18410.356,E2 18410.356} C_VEL
LIN {X 0,Y 414.148,Z 370.855,A -85,B 0,C 180,E1 18406.481,E2 18406.481} C_VEL
LIN {X 0,Y 412.179,Z 358.116,A -85,B 0,C 180,E1 18405.893,E2 18405.893} C_VEL
LIN {X 0,Y 401.332,Z 339.862,A -85,B 0,C 180,E1 18403.762,E2 18403.762} C_VEL
LIN {X 0,Y 390.818,Z 323.767,A -85,B 0,C 180,E1 18401.525,E2 18401.525} C_VEL
LIN {X 0,Y 389.24,Z 320.589,A -85,B 0,C 180,E1 18400.922,E2 18400.922} C_VEL
LIN {X 0,Y 383.515,Z 308.481,A -85,B 0,C 180,E1 18398.064,E2 18398.064} C_VEL
LIN {X 0,Y 378.922,Z 299.473,A -85,B 0,C 180,E1 18395.673,E2 18395.673} C_VEL
LIN {X 0,Y 376.959,Z 295.621,A -85,B 0,C 180,E1 18394.585,E2 18394.585} C_VEL
LIN {X 0,Y 374.481,Z 290.962,A -85,B 0,C 180,E1 18393.185,E2 18393.185} C_VEL
LIN {X 0,Y 372.529,Z 287.08,A -85,B 0,C 180,E1 18391.993,E2 18391.993} C_VEL
LIN {X 0,Y 370.011,Z 282.962,A -85,B 0,C 180,E1 18390.532,E2 18390.532} C_VEL
LIN {X 0,Y 369.766,Z 281.812,A -85,B 0,C 180,E1 18390.087,E2 18390.087} C_VEL
LIN {X 0,Y 369.74,Z 281.662,A -85,B 0,C 180,E1 18385.982,E2 18385.982} C_VEL
LIN {X 0,Y 369.743,Z 281.661,A -85,B 0,C 180,E1 18381.912,E2 18381.912} C_VEL
LIN {X 0,Y 369.739,Z 281.663,A -85,B 0,C 180,E1 18377.793,E2 18377.793} C_VEL
LIN {X 0,Y 369.739,Z 281.661,A -85,B 0,C 180,E1 18373.767,E2 18373.767} C_VEL
LIN {X 0,Y 369.734,Z 281.658,A -85,B 0,C 180,E1 18369.652,E2 18369.652} C_VEL
LIN {X 0,Y 369.733,Z 281.657,A -85,B 0,C 180,E1 18365.587,E2 18365.587} C_VEL
LIN {X 0,Y 369.736,Z 281.657,A -85,B 0,C 180,E1 18361.395,E2 18361.395} C_VEL
LIN {X 0,Y 369.727,Z 281.659,A -85,B 0,C 180,E1 18357.365,E2 18357.365} C_VEL
LIN {X 0,Y 369.724,Z 281.66,A -85,B 0,C 180,E1 18353.166,E2 18353.166} C_VEL
LIN {X 0,Y 369.706,Z 281.662,A -85,B 0,C 180,E1 18349.02,E2 18349.02} C_VEL
LIN {X 0,Y 369.699,Z 281.663,A -85,B 0,C 180,E1 18344.952,E2 18344.952} C_VEL
LIN {X 0,Y 369.702,Z 281.663,A -85,B 0,C 180,E1 18340.899,E2 18340.899} C_VEL
LIN {X 0,Y 369.709,Z 281.664,A -85,B 0,C 180,E1 18336.851,E2 18336.851} C_VEL
LIN {X 0,Y 369.755,Z 281.884,A -85,B 0,C 180,E1 18332.981,E2 18332.981} C_VEL
LIN {X 0,Y 371.134,Z 285.362,A -85,B 0,C 180,E1 18331.871,E2 18331.871} C_VEL
LIN {X 0,Y 372.683,Z 287.313,A -85,B 0,C 180,E1 18331.124,E2 18331.124} C_VEL
LIN {X 0,Y 374.511,Z 290.956,A -85,B 0,C 180,E1 18330.05,E2 18330.05} C_VEL
LIN {X 0,Y 375.692,Z 292.874,A -85,B 0,C 180,E1 18329.448,E2 18329.448} C_VEL
LIN {X 0,Y 378.566,Z 298.216,A -85,B 0,C 180,E1 18327.936,E2 18327.936} C_VEL
LIN {X 0,Y 383.546,Z 307.742,A -85,B 0,C 180,E1 18325.462,E2 18325.462} C_VEL
LIN {X 0,Y 388.247,Z 314.243,A -85,B 0,C 180,E1 18324.271,E2 18324.271} C_VEL
LIN {X 0,Y 400.17,Z 331.377,A -85,B 0,C 180,E1 18321.678,E2 18321.678} C_VEL
LIN {X 0,Y 411.289,Z 348.94,A -85,B 0,C 180,E1 18319.459,E2 18319.459} C_VEL
LIN {X 0,Y 417.201,Z 359.281,A -85,B 0,C 180,E1 18318.337,E2 18318.337} C_VEL
LIN {X 0,Y 408.529,Z 568.744,A -85,B 0,C 180,E1 18314.273,E2 18314.273} C_VEL
LIN {X 0,Y 406.756,Z 607.426,A -85,B 0,C 180,E1 18313.474,E2 18313.474} C_VEL
LIN {X 0,Y 404.738,Z 629.733,A -85,B 0,C 180,E1 18312.797,E2 18312.797} C_VEL
LIN {X 0,Y 402.257,Z 650.595,A -85,B 0,C 180,E1 18311.912,E2 18311.912} C_VEL
LIN {X 0,Y 399.115,Z 672.638,A -85,B 0,C 180,E1 18310.699,E2 18310.699} C_VEL
LIN {X 0,Y 395.842,Z 692.393,A -85,B 0,C 180,E1 18309.345,E2 18309.345} C_VEL
LIN {X 0,Y 392.231,Z 711.702,A -85,B 0,C 180,E1 18307.718,E2 18307.718} C_VEL
LIN {X 0,Y 388.546,Z 730.215,A -85,B 0,C 180,E1 18305.846,E2 18305.846} C_VEL
LIN {X 0,Y 384.778,Z 748.109,A -85,B 0,C 180,E1 18303.704,E2 18303.704} C_VEL
LIN {X 0,Y 381.164,Z 765.102,A -85,B 0,C 180,E1 18301.29,E2 18301.29} C_VEL
LIN {X 0,Y 377.779,Z 780.867,A -85,B 0,C 180,E1 18298.622,E2 18298.622} C_VEL
LIN {X 0,Y 374.995,Z 794.397,A -85,B 0,C 180,E1 18295.93,E2 18295.93} C_VEL
LIN {X 0,Y 372.641,Z 806.838,A -85,B 0,C 180,E1 18293.027,E2 18293.027} C_VEL
LIN {X 0,Y 370.823,Z 817.616,A -85,B 0,C 180,E1 18290.025,E2 18290.025} C_VEL
LIN {X 0,Y 369.472,Z 827.113,A -85,B 0,C 180,E1 18286.831,E2 18286.831} C_VEL
LIN {X 0,Y 368.632,Z 834.827,A -85,B 0,C 180,E1 18283.649,E2 18283.649} C_VEL
LIN {X 0,Y 368.197,Z 840.777,A -85,B 0,C 180,E1 18280.483,E2 18280.483} C_VEL
LIN {X 0,Y 368.024,Z 845.284,A -85,B 0,C 180,E1 18277.179,E2 18277.179} C_VEL
LIN {X 0,Y 367.98,Z 848.068,A -85,B 0,C 180,E1 18274.051,E2 18274.051} C_VEL
LIN {X 0,Y 367.995,Z 849.205,A -85,B 0,C 180,E1 18270.934,E2 18270.934} C_VEL
LIN {X 0,Y 367.987,Z 848.954,A -85,B 0,C 180,E1 18267.82,E2 18267.82} C_VEL
LIN {X 0,Y 367.992,Z 847.22,A -85,B 0,C 180,E1 18264.856,E2 18264.856} C_VEL
LIN {X 0,Y 368.06,Z 843.785,A -85,B 0,C 180,E1 18261.565,E2 18261.565} C_VEL
LIN {X 0,Y 368.294,Z 839.096,A -85,B 0,C 180,E1 18258.536,E2 18258.536} C_VEL
LIN {X 0,Y 368.874,Z 832.303,A -85,B 0,C 180,E1 18255.239,E2 18255.239} C_VEL
LIN {X 0,Y 369.879,Z 824.045,A -85,B 0,C 180,E1 18252.052,E2 18252.052} C_VEL
LIN {X 0,Y 371.436,Z 813.815,A -85,B 0,C 180,E1 18248.857,E2 18248.857} C_VEL
LIN {X 0,Y 373.497,Z 802.118,A -85,B 0,C 180,E1 18245.822,E2 18245.822} C_VEL
LIN {X 0,Y 376.073,Z 789.058,A -85,B 0,C 180,E1 18242.955,E2 18242.955} C_VEL
LIN {X 0,Y 379.1,Z 774.689,A -85,B 0,C 180,E1 18240.276,E2 18240.276} C_VEL
LIN {X 0,Y 382.482,Z 758.776,A -85,B 0,C 180,E1 18237.773,E2 18237.773} C_VEL
LIN {X 0,Y 386.188,Z 741.431,A -85,B 0,C 180,E1 18235.46,E2 18235.46} C_VEL
LIN {X 0,Y 389.959,Z 723.221,A -85,B 0,C 180,E1 18233.408,E2 18233.408} C_VEL
LIN {X 0,Y 393.517,Z 705.01,A -85,B 0,C 180,E1 18231.688,E2 18231.688} C_VEL
LIN {X 0,Y 397.032,Z 685.234,A -85,B 0,C 180,E1 18230.141,E2 18230.141} C_VEL
LIN {X 0,Y 400.267,Z 664.824,A -85,B 0,C 180,E1 18228.837,E2 18228.837} C_VEL
LIN {X 0,Y 403.136,Z 643.779,A -85,B 0,C 180,E1 18227.769,E2 18227.769} C_VEL
LIN {X 0,Y 405.463,Z 622.306,A -85,B 0,C 180,E1 18226.96,E2 18226.96} C_VEL
LIN {X 0,Y 407.199,Z 599.624,A -85,B 0,C 180,E1 18226.352,E2 18226.352} C_VEL
LIN {X 0,Y 416.029,Z 386.778,A -85,B 0,C 180,E1 18222.199,E2 18222.199} C_VEL
LIN {X 0,Y 417.055,Z 358.742,A -85,B 0,C 180,E1 18221.637,E2 18221.637} C_VEL
LIN {X 0,Y 405.918,Z 340.251,A -85,B 0,C 180,E1 18219.503,E2 18219.503} C_VEL
LIN {X 0,Y 394.791,Z 323.556,A -85,B 0,C 180,E1 18217.204,E2 18217.204} C_VEL
LIN {X 0,Y 385.207,Z 310.159,A -85,B 0,C 180,E1 18215.049,E2 18215.049} C_VEL
LIN {X 0,Y 383.354,Z 307.355,A -85,B 0,C 180,E1 18214.47,E2 18214.47} C_VEL
LIN {X 0,Y 379.694,Z 300.36,A -85,B 0,C 180,E1 18212.672,E2 18212.672} C_VEL
LIN {X 0,Y 377.203,Z 295.771,A -85,B 0,C 180,E1 18211.405,E2 18211.405} C_VEL
LIN {X 0,Y 374.775,Z 291.271,A -85,B 0,C 180,E1 18210.103,E2 18210.103} C_VEL
LIN {X 0,Y 372.838,Z 287.805,A -85,B 0,C 180,E1 18209.038,E2 18209.038} C_VEL
LIN {X 0,Y 372.02,Z 286.374,A -85,B 0,C 180,E1 18208.581,E2 18208.581} C_VEL
LIN {X 0,Y 370.076,Z 283.3,A -85,B 0,C 180,E1 18207.516,E2 18207.516} C_VEL
LIN {X 0,Y 369.751,Z 281.855,A -85,B 0,C 180,E1 18207.019,E2 18207.019} C_VEL
LIN {X 0,Y 369.728,Z 281.662,A -85,B 0,C 180,E1 18202.918,E2 18202.918} C_VEL
LIN {X 0,Y 369.718,Z 281.663,A -85,B 0,C 180,E1 18198.773,E2 18198.773} C_VEL
LIN {X 0,Y 369.725,Z 281.663,A -85,B 0,C 180,E1 18194.726,E2 18194.726} C_VEL
LIN {X 0,Y 369.71,Z 281.666,A -85,B 0,C 180,E1 18190.597,E2 18190.597} C_VEL
LIN {X 0,Y 369.721,Z 281.663,A -85,B 0,C 180,E1 18186.522,E2 18186.522} C_VEL
LIN {X 0,Y 369.719,Z 281.661,A -85,B 0,C 180,E1 18182.48,E2 18182.48} C_VEL
LIN {X 0,Y 369.728,Z 281.658,A -85,B 0,C 180,E1 18178.45,E2 18178.45} C_VEL
LIN {X 0,Y 369.729,Z 281.658,A -85,B 0,C 180,E1 18174.357,E2 18174.357} C_VEL
LIN {X 0,Y 369.733,Z 281.659,A -85,B 0,C 180,E1 18170.348,E2 18170.348} C_VEL
LIN {X 0,Y 369.738,Z 281.662,A -85,B 0,C 180,E1 18166.233,E2 18166.233} C_VEL
LIN {X 0,Y 369.737,Z 281.663,A -85,B 0,C 180,E1 18162.151,E2 18162.151} C_VEL
LIN {X 0,Y 369.74,Z 281.661,A -85,B 0,C 180,E1 18158.052,E2 18158.052} C_VEL
LIN {X 0,Y 369.737,Z 281.662,A -85,B 0,C 180,E1 18154.018,E2 18154.018} C_VEL
LIN {X 0,Y 369.751,Z 281.712,A -85,B 0,C 180,E1 18149.917,E2 18149.917} C_VEL
LIN {X 0,Y 369.895,Z 282.558,A -85,B 0,C 180,E1 18149.457,E2 18149.457} C_VEL
LIN {X 0,Y 371.596,Z 285.819,A -85,B 0,C 180,E1 18148.352,E2 18148.352} C_VEL
LIN {X 0,Y 372.696,Z 287.627,A -85,B 0,C 180,E1 18147.732,E2 18147.732} C_VEL
LIN {X 0,Y 374.904,Z 291.48,A -85,B 0,C 180,E1 18146.491,E2 18146.491} C_VEL
LIN {X 0,Y 377.396,Z 296.189,A -85,B 0,C 180,E1 18145.092,E2 18145.092} C_VEL
LIN {X 0,Y 382.565,Z 306.63,A -85,B 0,C 180,E1 18142.296,E2 18142.296} C_VEL
LIN {X 0,Y 388.095,Z 318.16,A -85,B 0,C 180,E1 18139.516,E2 18139.516} C_VEL
LIN {X 0,Y 390.693,Z 323.6,A -85,B 0,C 180,E1 18138.386,E2 18138.386} C_VEL
LIN {X 0,Y 401.953,Z 340.86,A -85,B 0,C 180,E1 18136.002,E2 18136.002} C_VEL
LIN {X 0,Y 412.338,Z 358.489,A -85,B 0,C 180,E1 18133.968,E2 18133.968} C_VEL
LIN {X 0,Y 414.103,Z 372.276,A -85,B 0,C 180,E1 18133.386,E2 18133.386} C_VEL
LIN {X 0,Y 406.534,Z 595.323,A -85,B 0,C 180,E1 18129.368,E2 18129.368} C_VEL
LIN {X 0,Y 404.942,Z 616.02,A -85,B 0,C 180,E1 18128.763,E2 18128.763} C_VEL
LIN {X 0,Y 402.776,Z 635.72,A -85,B 0,C 180,E1 18127.948,E2 18127.948} C_VEL
LIN {X 0,Y 399.989,Z 655.587,A -85,B 0,C 180,E1 18126.864,E2 18126.864} C_VEL
LIN {X 0,Y 396.893,Z 674.054,A -85,B 0,C 180,E1 18125.586,E2 18125.586} C_VEL
LIN {X 0,Y 393.329,Z 692.461,A -85,B 0,C 180,E1 18124.003,E2 18124.003} C_VEL
LIN {X 0,Y 389.545,Z 709.734,A -85,B 0,C 180,E1 18122.18,E2 18122.18} C_VEL
LIN {X 0,Y 385.851,Z 725.451,A -85,B 0,C 180,E1 18120.179,E2 18120.179} C_VEL
LIN {X 0,Y 382.184,Z 740.266,A -85,B 0,C 180,E1 18117.923,E2 18117.923} C_VEL
LIN {X 0,Y 378.832,Z 753.668,A -85,B 0,C 180,E1 18115.48,E2 18115.48} C_VEL
LIN {X 0,Y 375.68,Z 766.324,A -85,B 0,C 180,E1 18112.7,E2 18112.7} C_VEL
LIN {X 0,Y 373.055,Z 777.329,A -85,B 0,C 180,E1 18109.736,E2 18109.736} C_VEL
LIN {X 0,Y 371.111,Z 786.231,A -85,B 0,C 180,E1 18106.788,E2 18106.788} C_VEL
LIN {X 0,Y 369.562,Z 789.263,A -85,B 0,C 180,E1 18105.706,E2 18105.706} C_VEL
LIN {X 0,Y 362.175,Z 796.546,A -85,B 0,C 180,E1 18102.796,E2 18102.796} C_VEL
LIN {X 0,Y 361.143,Z 798.41,A -85,B 0,C 180,E1 18101.796,E2 18101.796} C_VEL
LIN {X 0,Y 360.49,Z 803.312,A -85,B 0,C 180,E1 18098.453,E2 18098.453} C_VEL
LIN {X 0,Y 360.183,Z 806.576,A -85,B 0,C 180,E1 18095.096,E2 18095.096} C_VEL
LIN {X 0,Y 360.087,Z 808.211,A -85,B 0,C 180,E1 18091.909,E2 18091.909} C_VEL
LIN {X 0,Y 360.074,Z 808.326,A -85,B 0,C 180,E1 18088.727,E2 18088.727} C_VEL
LIN {X 0,Y 360.156,Z 806.914,A -85,B 0,C 180,E1 18085.311,E2 18085.311} C_VEL
LIN {X 0,Y 360.415,Z 804.012,A -85,B 0,C 180,E1 18082.027,E2 18082.027} C_VEL
LIN {X 0,Y 360.975,Z 799.649,A -85,B 0,C 180,E1 18078.82,E2 18078.82} C_VEL
LIN {X 0,Y 361.982,Z 793.579,A -85,B 0,C 180,E1 18075.606,E2 18075.606} C_VEL
LIN {X 0,Y 363.583,Z 785.754,A -85,B 0,C 180,E1 18072.393,E2 18072.393} C_VEL
LIN {X 0,Y 365.925,Z 775.798,A -85,B 0,C 180,E1 18069.146,E2 18069.146} C_VEL
LIN {X 0,Y 368.796,Z 764.548,A -85,B 0,C 180,E1 18066.175,E2 18066.175} C_VEL
LIN {X 0,Y 372.088,Z 752.211,A -85,B 0,C 180,E1 18063.486,E2 18063.486} C_VEL
LIN {X 0,Y 375.689,Z 738.636,A -85,B 0,C 180,E1 18061.029,E2 18061.029} C_VEL
LIN {X 0,Y 379.46,Z 723.948,A -85,B 0,C 180,E1 18058.818,E2 18058.818} C_VEL
LIN {X 0,Y 383.39,Z 707.836,A -85,B 0,C 180,E1 18056.794,E2 18056.794} C_VEL
LIN {X 0,Y 387.219,Z 690.859,A -85,B 0,C 180,E1 18055.025,E2 18055.025} C_VEL
LIN {X 0,Y 390.805,Z 673.103,A -85,B 0,C 180,E1 18053.5,E2 18053.5} C_VEL
LIN {X 0,Y 394.05,Z 654.329,A -85,B 0,C 180,E1 18052.21,E2 18052.21} C_VEL
LIN {X 0,Y 396.768,Z 635.388,A -85,B 0,C 180,E1 18051.183,E2 18051.183} C_VEL
LIN {X 0,Y 399.053,Z 615.083,A -85,B 0,C 180,E1 18050.348,E2 18050.348} C_VEL
LIN {X 0,Y 400.666,Z 594.597,A -85,B 0,C 180,E1 18049.757,E2 18049.757} C_VEL
